// TIA Portal V20 export
// export: Created 2025-12-01T14:57:26.0447833Z, ExportSetting None, DisplayName Totally Integrated Automation Portal, DisplayVersion V20 Update 3, DisplayName TIA Portal Openness, DisplayVersion V20 Update 3, DisplayName TIA Portal Version Control Interface, DisplayVersion V20 Update 3, DisplayName STEP 7 Professional, DisplayVersion V20 Update 3, DisplayName STEP 7 Safety, DisplayVersion V20 Update 2, DisplayName WinCC Basic/Comfort/Advanced, DisplayVersion V20 Update 3, DisplayName WinCC Professional, DisplayVersion V20 Update 3, DisplayName WinCC Unified, DisplayVersion V20 Update 3
FUNCTION_BLOCK "FB454_CRTL_FRAT_E1_S2S3S4"   // FB454, LAD
TITLE = Control del Ramal de Salidas
{ S7_Optimized_Access := 'FALSE' }
AUTHOR : TLigero
NAME : 20190911
VERSION : 3.5
// stored: AutoNumber false, SetENOAutomatically false
   VAR_INPUT
      Mesa : UInt;   // Número de mesa
      En_Tension : Bool;
      pHsMx_E1 : Bool;   // pHs de ausencia de la Mesa por E1
      pHsMx_S2 : Bool;   // pHs de ausencia de la Mesa por S2
      pHsMx_S3 : Bool;   // pHs de ausencia de la Mesa por S3
      pHsMx_S4 : Bool;
      pHsMx_Pres : Bool;
      PosTR_E1S3 : Bool;   // Posicion del TR en E1E3
      PosTR_S2S4 : Bool;   // Posicion del TR en E2E4
      Termico_E1S3 : Bool;   // Proteccion del Tx en E1E3
      Termico_S2S4 : Bool;   // Proteccion del Tx en E2E4
      Avance_E1 : Bool;   // Avance del Tx en E1E3
      Avance_S2 : Bool;   // Avance del Tx en E2E4
      PTF_Sal_M2 : Bool;   // S2 >> Mesa Siguiente PTF
      NXT_Avance_S2 : Bool;   // S2 >> Mesa Siguiente avanzando
      PTF_Sal_M3 : Bool;   // S3 >> Mesa Siguiente PTF
      NXT_Avance_S3 : Bool;   // S3 >> Mesa Siguiente avanzando
      PTF_Sal_M4 : Bool;   // S2 >> Mesa Siguiente PTF
      NXT_Avance_S4 : Bool;   // S2 >> Mesa Siguiente avanzando
      F_EnvMens_Mx : Bool;   // Fin de Envio de Mensaje
      Salida_S2S4_Ausencia : Bool;   // True por ausencia. false por presencia
      Mx_BloqActivo_S2 : Bool;   // Bloqueo Activo de la Mesa
      Mx_FlujoPrin_S2 : Bool;   // El flujo principal es Saliendo por S2
      Mx_BloqActivo_S4 : Bool;   // Bloqueo Activo de la Mesa
      Mx_FlujoPrin_S4 : Bool;   // El flujo principal es Saliendo por S2
      AVTF_MAnt_Mx : Bool;   // E1 >> Mesa Anterior AVTF
      Simul_Mx : Bool;   // Activar simultaneo de mesa
      Num_Cruce : UInt;   // Número de cruce.
      DB_FIFO_Cruce : UInt := 213;   // DB de la FIFO de ordenes del cruce
      Long_FIFO_Cruce : UInt := 1;   // Longitut de la FIFO de ordenes del cruce
      ValorOrden_S2 : Word := 16#81;   // Con que orden entra por S2
      ValorOrden_S4 : Word := 16#81;   // Con que orden entra por S2
      MesaS2 : UInt;   // Número de mesa por S2
      MesaS3 : UInt;   // Número de mesa por S3
      MesaS4 : UInt;   // Número de mesa por S3
      V_CNT_ApHsMx_E1 : UDInt;   // Valor de Ausencia por E1 en ms
      V_CNT_ApHsMx_S2 : UDInt;   // Valor de Ausencia por S2 en ms
      V_CNT_ApHsMx_S3 : UDInt;   // Valor de Ausencia por S3 en ms
      V_CNT_ApHsMx_S4 : UDInt;   // Valor de Ausencia por S3 en ms
      V_CNT_SIMUL_S3 : UDInt;   // Valor de ventana para iniciar simultanero por S3 en ms
      V_Vaciado : UDInt := 15000;   // Valor de vaciado en ms
      V_TOut_Tx_Mx : UDInt := 15000;   // TimeOut de Atasco en ms
      V_TOut_TR : UDInt := 5000;   // TimeOut de Transfer en ms
   END_VAR
   VAR_OUTPUT
      P_EnvMens_PMx : Bool;   // Permiso de Enviar Mensaje de Presencia
      Etiqueta_Jdt : ULInt;   // Etiqueta que ha sido leida
      Orden_Ejecutada_Jdt : UInt;   // Orden que se ha ejecutado
      PTF_MAnt_Mx : Bool;   // E1 >> Mesa Anterior PTF
      AVTF_Sal_M2 : Bool;   // S2 >> Mesa Siguiente AVTF
      AVTF_Sal_M3 : Bool;   // S3 >> Mesa Siguiente AVTF
      AVTF_Sal_M4 : Bool;   // S3 >> Mesa Siguiente AVTF
   END_VAR
   VAR
      T1_ET00 : Bool;
      T1_ET01 : Bool;
      T1_ET02 : Bool;
      T1_ET03 : Bool;
      T1_ET10 : Bool;
      T1_ET11 : Bool;
      T1_ET12 : Bool;
      T1_ET50 : Bool;
      T1_ET60 : Bool;
      T1_ET80 : Bool;
      T1_ET70 : Bool;
      T1_ET110 : Bool;
      T1_ET111 : Bool;
      T1_ET112 : Bool;
      FIFO_OK : Bool;
      TRANS_OK : Bool;
      O_Bloqueo : Bool;
      Err_Detec_PHS : Bool;
      FN_ET02 : Bool;
      MemFN_pHsE1 : Bool;
      MemFN_pHsS3 : Bool;
      MemFN_pHsS2 : Bool;
      MemFN_pHsS4 : Bool;
      MemAuxFN_pHsE1 : Bool;
      MemAuxFN_pHsS3 : Bool;
      MemAuxFN_pHsS2 : Bool;
      MemAuxFN_pHsS4 : Bool;
      OK_TmpAusE1 : Bool;
      OK_TmpAusS3 : Bool;
      OK_TmpAusS2 : Bool;
      OK_TmpAusS4 : Bool;
      OK_Tmp_Paro : Bool;
      OK_Tmp_Simul : Bool;
      maux_fp_disparo : Bool;
      vaciado_ok { ExternalAccessible := 'False'; ExternalVisible := 'False'; ExternalWritable := 'False'} : Bool;
      Fin_reposicionamiento : Bool;
      Maux_reposicionamiento : Bool;
      CNT_Seguridad_E1 { ExternalAccessible := 'False'; ExternalVisible := 'False'; ExternalWritable := 'False'} : Bool;
      Mem_Motor_E1_Ha_Parado_NoHayPTFS2 : Bool;   // No hay permiso de transferencia a la salida por 2, por tanto cuando se reanude la secuencia a Etapa 60, no poner en marcha El motor E1
      Reposicionamiento_ok : Bool;
      TmpAus_E1 : UDInt;
      TmpAus_S2 : UDInt;
      TmpAus_S3 : UDInt;
      TmpAus_S4 : UDInt;
      TmpSeg_E1 : UDInt;
      Tmp_Paro : UDInt;
      Tmp_Simul_S3 : UDInt;
      TOUT_TR_PosS2 : UDInt;
      TOUT_TR_PosE1S3 : UDInt;
      TIM_Vaciado : UDInt;
      TOUT_E1S3 : UDInt;
      TOUT_S2 : UDInt;
      TMP_Reposicionamiento : UDInt;
      Tout_tope : UDInt;
      TMP_RearmePosicionamiento : UDInt;
      Datos_Scanner { S7_SetPoint := 'True'} : "ROUT_Orden_Fifo_Scanner";
   END_VAR
   VAR_TEMP
      O_Sal_S3 : Bool;
      O_Sal_S2 : Bool;
      O_Sal_S4 : Bool;
      O_Vaciar : Bool;
      Moti_ERRO : Bool;
      Moti_NENC : Bool;
      Moti_NORM : Bool;
      Moti_INIC : Bool;
      tout_ir_s2 : Bool;
      tout_ir_s3 : Bool;
      atasco : Bool;
      timeout_s2 : Bool;
      Tout_tope_Q : Bool;
      Aux_W_Moti : Word;
      INT_ORDEN : UInt;
      Aux_W_Orden : Word;
      I_Ord_Filtrada : UInt;
      I_V_Ord_S2 : UInt;
      I_V_Ord_S4 : UInt;
   END_VAR
   VAR_TEMP   // added for the SCL form of the ladder/FBD networks
      _w1 : Bool;
      _w2 : Bool;
      _w3 : Bool;
      _w4 : Bool;
      _w5 : Bool;
      _w6 : Bool;
   END_VAR
BEGIN

REGION Network 1: Reset Error Mesa y estado manual
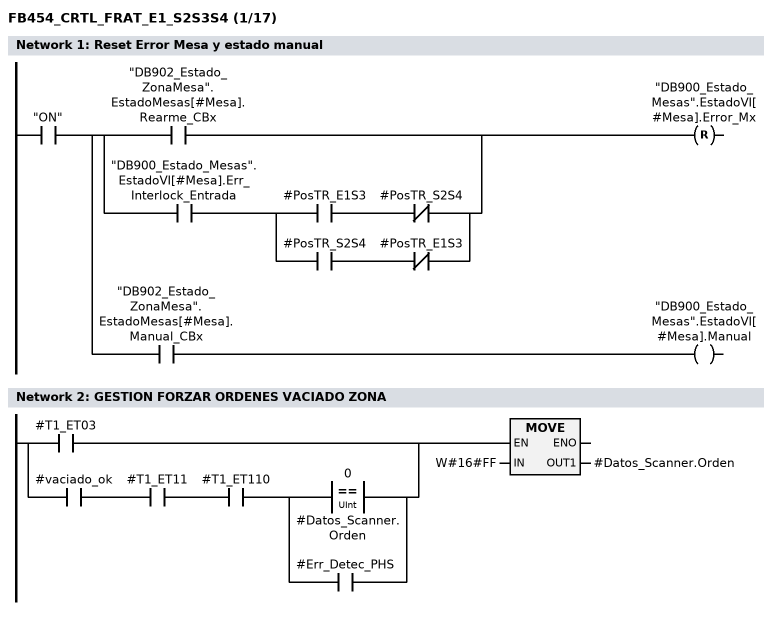
   RUNG wire#powerrail
      Contact( "ON" )
      wire#w1
      Contact( "DB902_Estado_ZonaMesa".EstadoMesas[#Mesa].Rearme_CBx )
      wire#w2
      R_Coil( "DB900_Estado_Mesas".EstadoVI[#Mesa].Error_Mx )
   END_RUNG
   RUNG wire#w1
      Contact( "DB900_Estado_Mesas".EstadoVI[#Mesa].Err_Interlock_Entrada )
      wire#w3
      Contact( #PosTR_E1S3 )
      I_Contact( #PosTR_S2S4 )
   END_RUNG wire#w2
   RUNG wire#w3
      Contact( #PosTR_S2S4 )
      I_Contact( #PosTR_E1S3 )
   END_RUNG wire#w2
   RUNG wire#w1
      Contact( "DB902_Estado_ZonaMesa".EstadoMesas[#Mesa].Manual_CBx )
      Coil( "DB900_Estado_Mesas".EstadoVI[#Mesa].Manual )
   END_RUNG
   // the same network as SCL:
   IF "ON" AND ("DB902_Estado_ZonaMesa".EstadoMesas[#Mesa].Rearme_CBx OR ("DB900_Estado_Mesas".EstadoVI[#Mesa].Err_Interlock_Entrada AND ((#PosTR_E1S3 AND NOT #PosTR_S2S4) OR (#PosTR_S2S4 AND NOT #PosTR_E1S3)))) THEN
       "DB900_Estado_Mesas".EstadoVI[#Mesa].Error_Mx := FALSE;
   END_IF;
   "DB900_Estado_Mesas".EstadoVI[#Mesa].Manual := "ON" AND "DB902_Estado_ZonaMesa".EstadoMesas[#Mesa].Manual_CBx;
END_REGION

REGION Network 2: GESTION FORZAR ORDENES VACIADO ZONA
   RUNG wire#powerrail
      Contact( #T1_ET03 )
      wire#w1
      { S7_GenerateENO := "TRUE" } Move(in := W#16#FF, out1 => #Datos_Scanner.Orden)
   END_RUNG
   RUNG wire#powerrail
      Contact( #vaciado_ok )
      Contact( #T1_ET11 )
      Contact( #T1_ET110 )
      wire#w2
      { S7_Templates := "SrcType := UInt" } EQ_Contact(in1 := 0, in2 := #Datos_Scanner.Orden)
   END_RUNG wire#w1
   RUNG wire#w2
      Contact( #Err_Detec_PHS )
   END_RUNG wire#w1
   // the same network as SCL:
   IF #T1_ET03 OR (#vaciado_ok AND #T1_ET11 AND #T1_ET110 AND ((0 = #Datos_Scanner.Orden) OR #Err_Detec_PHS)) THEN
       #Datos_Scanner.Orden := W#16#FF;
   END_IF;
END_REGION

REGION Network 3: Extraer orden
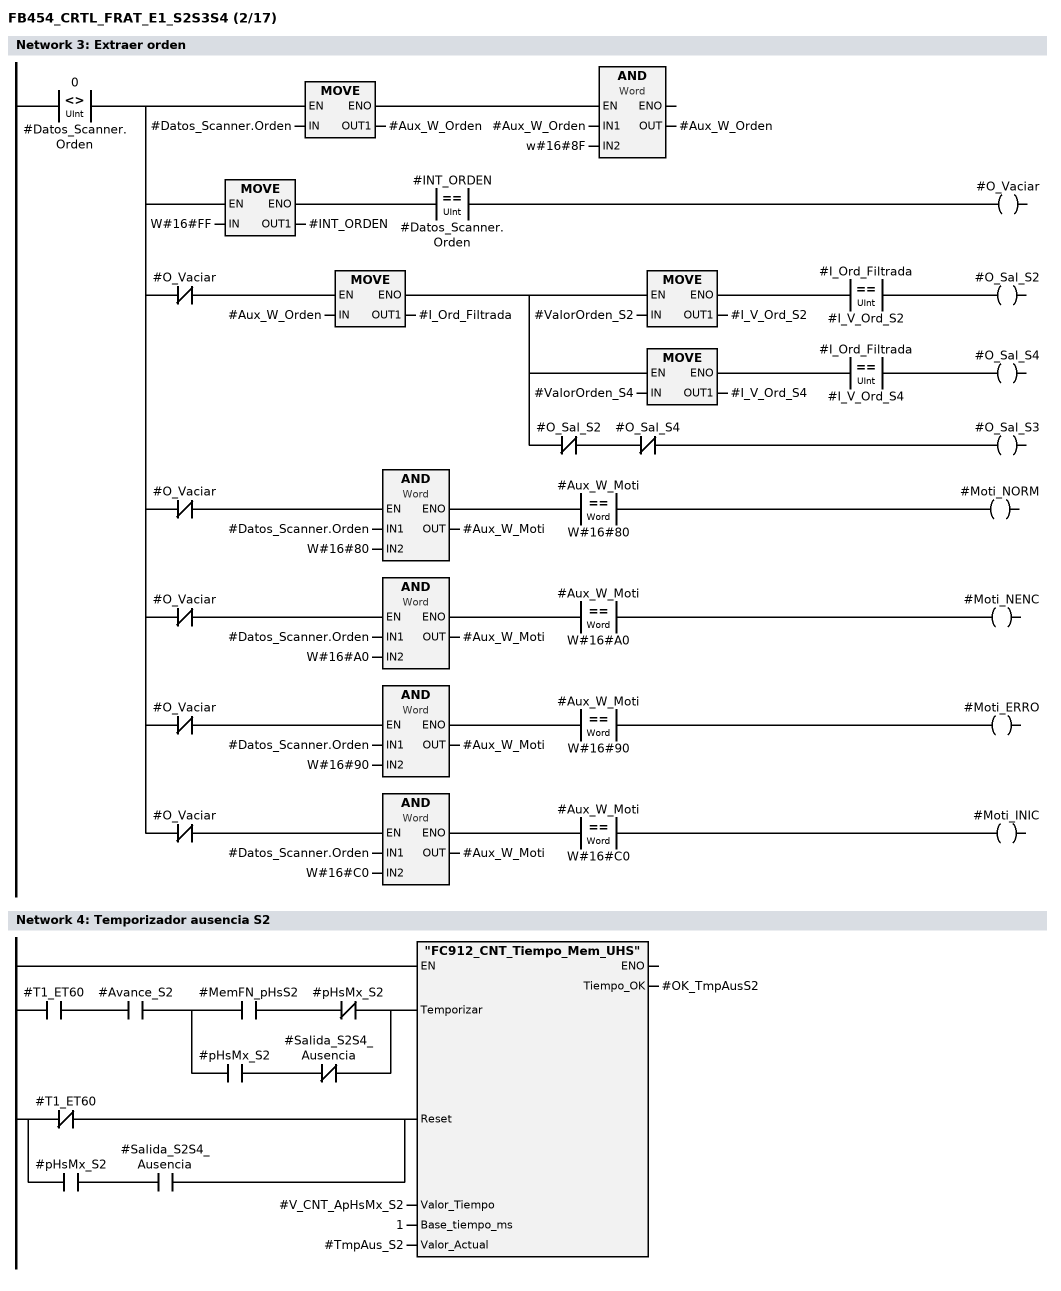
   RUNG wire#powerrail
      { S7_Templates := "SrcType := UInt" } NE_Contact(in1 := 0, in2 := #Datos_Scanner.Orden)
      wire#w1
      { S7_GenerateENO := "TRUE" } Move(in := #Datos_Scanner.Orden, out1 => #Aux_W_Orden)
      { S7_Templates := "SrcType := Word"; S7_GenerateENO := "TRUE" } And(in1 := #Aux_W_Orden, in2 := w#16#8F, out => #Aux_W_Orden)
   END_RUNG
   RUNG wire#w1
      { S7_GenerateENO := "TRUE" } Move(in := W#16#FF, out1 => #INT_ORDEN)
      { S7_Templates := "SrcType := UInt" } EQ_Contact(in1 := #INT_ORDEN, in2 := #Datos_Scanner.Orden)
      Coil( #O_Vaciar )
   END_RUNG
   RUNG wire#w1
      I_Contact( #O_Vaciar )
      { S7_GenerateENO := "TRUE" } Move(in := #Aux_W_Orden, out1 => #I_Ord_Filtrada)
      wire#w2
      { S7_GenerateENO := "TRUE" } Move(in := #ValorOrden_S2, out1 => #I_V_Ord_S2)
      { S7_Templates := "SrcType := UInt" } EQ_Contact(in1 := #I_Ord_Filtrada, in2 := #I_V_Ord_S2)
      Coil( #O_Sal_S2 )
   END_RUNG
   RUNG wire#w2
      { S7_GenerateENO := "TRUE" } Move(in := #ValorOrden_S4, out1 => #I_V_Ord_S4)
      { S7_Templates := "SrcType := UInt" } EQ_Contact(in1 := #I_Ord_Filtrada, in2 := #I_V_Ord_S4)
      Coil( #O_Sal_S4 )
   END_RUNG
   RUNG wire#w2
      I_Contact( #O_Sal_S2 )
      I_Contact( #O_Sal_S4 )
      Coil( #O_Sal_S3 )
   END_RUNG
   RUNG wire#w1
      I_Contact( #O_Vaciar )
      { S7_Templates := "SrcType := Word"; S7_GenerateENO := "TRUE" } And(in1 := #Datos_Scanner.Orden, in2 := W#16#80, out => #Aux_W_Moti)
      { S7_Templates := "SrcType := Word" } EQ_Contact(in1 := #Aux_W_Moti, in2 := W#16#80)
      Coil( #Moti_NORM )
   END_RUNG
   RUNG wire#w1
      I_Contact( #O_Vaciar )
      { S7_Templates := "SrcType := Word"; S7_GenerateENO := "TRUE" } And(in1 := #Datos_Scanner.Orden, in2 := W#16#A0, out => #Aux_W_Moti)
      { S7_Templates := "SrcType := Word" } EQ_Contact(in1 := #Aux_W_Moti, in2 := W#16#A0)
      Coil( #Moti_NENC )
   END_RUNG
   RUNG wire#w1
      I_Contact( #O_Vaciar )
      { S7_Templates := "SrcType := Word"; S7_GenerateENO := "TRUE" } And(in1 := #Datos_Scanner.Orden, in2 := W#16#90, out => #Aux_W_Moti)
      { S7_Templates := "SrcType := Word" } EQ_Contact(in1 := #Aux_W_Moti, in2 := W#16#90)
      Coil( #Moti_ERRO )
   END_RUNG
   RUNG wire#w1
      I_Contact( #O_Vaciar )
      { S7_Templates := "SrcType := Word"; S7_GenerateENO := "TRUE" } And(in1 := #Datos_Scanner.Orden, in2 := W#16#C0, out => #Aux_W_Moti)
      { S7_Templates := "SrcType := Word" } EQ_Contact(in1 := #Aux_W_Moti, in2 := W#16#C0)
      Coil( #Moti_INIC )
   END_RUNG
   // the same network as SCL:
   // ENO of a box is taken as its EN; it also drops when the box reports an error
   #_w1 := 0 <> #Datos_Scanner.Orden;
   IF #_w1 THEN
       #Aux_W_Orden := #Datos_Scanner.Orden;
       #Aux_W_Orden := #Aux_W_Orden AND w#16#8F;
       #INT_ORDEN := W#16#FF;
   END_IF;
   #O_Vaciar := #_w1 AND (#INT_ORDEN = #Datos_Scanner.Orden);
   #_w2 := #_w1 AND NOT #O_Vaciar;
   IF #_w2 THEN
       #I_Ord_Filtrada := #Aux_W_Orden;
       #I_V_Ord_S2 := #ValorOrden_S2;
   END_IF;
   #O_Sal_S2 := #_w2 AND (#I_Ord_Filtrada = #I_V_Ord_S2);
   IF #_w2 THEN #I_V_Ord_S4 := #ValorOrden_S4; END_IF;
   #O_Sal_S4 := #_w2 AND (#I_Ord_Filtrada = #I_V_Ord_S4);
   #O_Sal_S3 := #_w2 AND NOT #O_Sal_S2 AND NOT #O_Sal_S4;
   #_w3 := #_w1 AND NOT #O_Vaciar;
   IF #_w3 THEN #Aux_W_Moti := #Datos_Scanner.Orden AND W#16#80; END_IF;
   #Moti_NORM := #_w3 AND (#Aux_W_Moti = W#16#80);
   #_w4 := #_w1 AND NOT #O_Vaciar;
   IF #_w4 THEN #Aux_W_Moti := #Datos_Scanner.Orden AND W#16#A0; END_IF;
   #Moti_NENC := #_w4 AND (#Aux_W_Moti = W#16#A0);
   #_w5 := #_w1 AND NOT #O_Vaciar;
   IF #_w5 THEN #Aux_W_Moti := #Datos_Scanner.Orden AND W#16#90; END_IF;
   #Moti_ERRO := #_w5 AND (#Aux_W_Moti = W#16#90);
   #_w6 := #_w1 AND NOT #O_Vaciar;
   IF #_w6 THEN #Aux_W_Moti := #Datos_Scanner.Orden AND W#16#C0; END_IF;
   #Moti_INIC := #_w6 AND (#Aux_W_Moti = W#16#C0);
END_REGION

REGION Network 4: Temporizador ausencia S2
   RUNG wire#powerrail
      "FC912_CNT_Tiempo_Mem_UHS"(Temporizar := wire#w2, Reset := wire#w3, Valor_Tiempo := #V_CNT_ApHsMx_S2, Base_tiempo_ms := 1, Valor_Actual := #TmpAus_S2, Tiempo_OK => #OK_TmpAusS2)
   END_RUNG
   RUNG wire#powerrail
      Contact( #T1_ET60 )
      Contact( #Avance_S2 )
      wire#w1
      Contact( #MemFN_pHsS2 )
      I_Contact( #pHsMx_S2 )
   END_RUNG wire#w2
   RUNG wire#w1
      Contact( #pHsMx_S2 )
      I_Contact( #Salida_S2S4_Ausencia )
   END_RUNG wire#w2
   RUNG wire#powerrail
      I_Contact( #T1_ET60 )
   END_RUNG wire#w3
   RUNG wire#powerrail
      Contact( #pHsMx_S2 )
      Contact( #Salida_S2S4_Ausencia )
   END_RUNG wire#w3
   // the same network as SCL:
   "FC912_CNT_Tiempo_Mem_UHS"(Temporizar := #T1_ET60 AND #Avance_S2 AND ((#MemFN_pHsS2 AND NOT #pHsMx_S2) OR (#pHsMx_S2 AND NOT #Salida_S2S4_Ausencia)),
                           Reset := NOT #T1_ET60 OR (#pHsMx_S2 AND #Salida_S2S4_Ausencia),
                           Valor_Tiempo := #V_CNT_ApHsMx_S2,
                           Base_tiempo_ms := 1,
                           Valor_Actual := #TmpAus_S2,
                           Tiempo_OK => #OK_TmpAusS2);
END_REGION

REGION Network 5: Temporizador ausencia S4
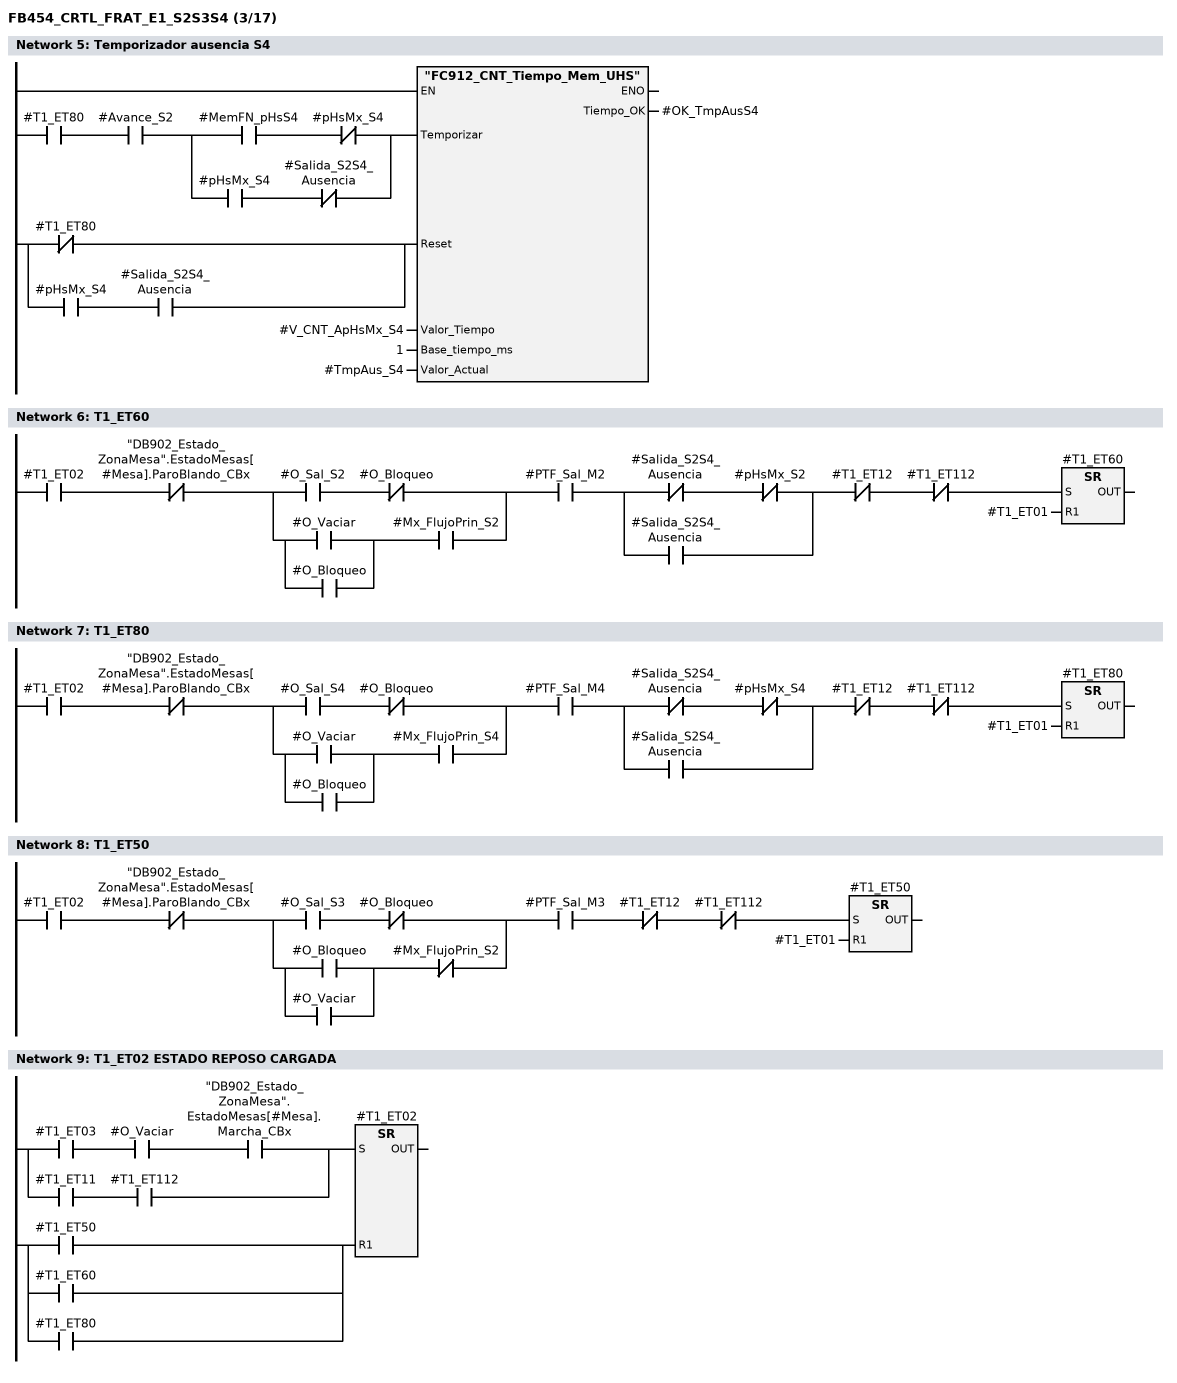
   RUNG wire#powerrail
      "FC912_CNT_Tiempo_Mem_UHS"(Temporizar := wire#w2, Reset := wire#w3, Valor_Tiempo := #V_CNT_ApHsMx_S4, Base_tiempo_ms := 1, Valor_Actual := #TmpAus_S4, Tiempo_OK => #OK_TmpAusS4)
   END_RUNG
   RUNG wire#powerrail
      Contact( #T1_ET80 )
      Contact( #Avance_S2 )
      wire#w1
      Contact( #MemFN_pHsS4 )
      I_Contact( #pHsMx_S4 )
   END_RUNG wire#w2
   RUNG wire#w1
      Contact( #pHsMx_S4 )
      I_Contact( #Salida_S2S4_Ausencia )
   END_RUNG wire#w2
   RUNG wire#powerrail
      I_Contact( #T1_ET80 )
   END_RUNG wire#w3
   RUNG wire#powerrail
      Contact( #pHsMx_S4 )
      Contact( #Salida_S2S4_Ausencia )
   END_RUNG wire#w3
   // the same network as SCL:
   "FC912_CNT_Tiempo_Mem_UHS"(Temporizar := #T1_ET80 AND #Avance_S2 AND ((#MemFN_pHsS4 AND NOT #pHsMx_S4) OR (#pHsMx_S4 AND NOT #Salida_S2S4_Ausencia)),
                           Reset := NOT #T1_ET80 OR (#pHsMx_S4 AND #Salida_S2S4_Ausencia),
                           Valor_Tiempo := #V_CNT_ApHsMx_S4,
                           Base_tiempo_ms := 1,
                           Valor_Actual := #TmpAus_S4,
                           Tiempo_OK => #OK_TmpAusS4);
END_REGION

REGION Network 6: T1_ET60
   RUNG wire#powerrail
      Contact( #T1_ET02 )
      I_Contact( "DB902_Estado_ZonaMesa".EstadoMesas[#Mesa].ParoBlando_CBx )
      wire#w1
      Contact( #O_Sal_S2 )
      I_Contact( #O_Bloqueo )
      wire#w2
      Contact( #PTF_Sal_M2 )
      wire#w4
      I_Contact( #Salida_S2S4_Ausencia )
      I_Contact( #pHsMx_S2 )
      wire#w5
      I_Contact( #T1_ET12 )
      I_Contact( #T1_ET112 )
      S_SR(operand := #T1_ET60, r1 := #T1_ET01)
   END_RUNG
   RUNG wire#w1
      Contact( #O_Vaciar )
      wire#w3
      Contact( #Mx_FlujoPrin_S2 )
   END_RUNG wire#w2
   RUNG wire#w1
      Contact( #O_Bloqueo )
   END_RUNG wire#w3
   RUNG wire#w4
      Contact( #Salida_S2S4_Ausencia )
   END_RUNG wire#w5
   // the same network as SCL:
   IF #T1_ET02 AND NOT "DB902_Estado_ZonaMesa".EstadoMesas[#Mesa].ParoBlando_CBx AND ((#O_Sal_S2 AND NOT #O_Bloqueo) OR ((#O_Vaciar OR #O_Bloqueo) AND #Mx_FlujoPrin_S2)) AND #PTF_Sal_M2 AND ((NOT #Salida_S2S4_Ausencia AND NOT #pHsMx_S2) OR #Salida_S2S4_Ausencia) AND NOT #T1_ET12 AND NOT #T1_ET112 THEN
       #T1_ET60 := TRUE;   // SR flip-flop
   END_IF;
   IF #T1_ET01 THEN #T1_ET60 := FALSE; END_IF;
END_REGION

REGION Network 7: T1_ET80
   RUNG wire#powerrail
      Contact( #T1_ET02 )
      I_Contact( "DB902_Estado_ZonaMesa".EstadoMesas[#Mesa].ParoBlando_CBx )
      wire#w1
      Contact( #O_Sal_S4 )
      I_Contact( #O_Bloqueo )
      wire#w2
      Contact( #PTF_Sal_M4 )
      wire#w4
      I_Contact( #Salida_S2S4_Ausencia )
      I_Contact( #pHsMx_S4 )
      wire#w5
      I_Contact( #T1_ET12 )
      I_Contact( #T1_ET112 )
      S_SR(operand := #T1_ET80, r1 := #T1_ET01)
   END_RUNG
   RUNG wire#w1
      Contact( #O_Vaciar )
      wire#w3
      Contact( #Mx_FlujoPrin_S4 )
   END_RUNG wire#w2
   RUNG wire#w1
      Contact( #O_Bloqueo )
   END_RUNG wire#w3
   RUNG wire#w4
      Contact( #Salida_S2S4_Ausencia )
   END_RUNG wire#w5
   // the same network as SCL:
   IF #T1_ET02 AND NOT "DB902_Estado_ZonaMesa".EstadoMesas[#Mesa].ParoBlando_CBx AND ((#O_Sal_S4 AND NOT #O_Bloqueo) OR ((#O_Vaciar OR #O_Bloqueo) AND #Mx_FlujoPrin_S4)) AND #PTF_Sal_M4 AND ((NOT #Salida_S2S4_Ausencia AND NOT #pHsMx_S4) OR #Salida_S2S4_Ausencia) AND NOT #T1_ET12 AND NOT #T1_ET112 THEN
       #T1_ET80 := TRUE;   // SR flip-flop
   END_IF;
   IF #T1_ET01 THEN #T1_ET80 := FALSE; END_IF;
END_REGION

REGION Network 8: T1_ET50
   RUNG wire#powerrail
      Contact( #T1_ET02 )
      I_Contact( "DB902_Estado_ZonaMesa".EstadoMesas[#Mesa].ParoBlando_CBx )
      wire#w1
      Contact( #O_Sal_S3 )
      I_Contact( #O_Bloqueo )
      wire#w2
      Contact( #PTF_Sal_M3 )
      I_Contact( #T1_ET12 )
      I_Contact( #T1_ET112 )
      S_SR(operand := #T1_ET50, r1 := #T1_ET01)
   END_RUNG
   RUNG wire#w1
      Contact( #O_Bloqueo )
      wire#w3
      I_Contact( #Mx_FlujoPrin_S2 )
   END_RUNG wire#w2
   RUNG wire#w1
      Contact( #O_Vaciar )
   END_RUNG wire#w3
   // the same network as SCL:
   IF #T1_ET02 AND NOT "DB902_Estado_ZonaMesa".EstadoMesas[#Mesa].ParoBlando_CBx AND ((#O_Sal_S3 AND NOT #O_Bloqueo) OR ((#O_Bloqueo OR #O_Vaciar) AND NOT #Mx_FlujoPrin_S2)) AND #PTF_Sal_M3 AND NOT #T1_ET12 AND NOT #T1_ET112 THEN
       #T1_ET50 := TRUE;   // SR flip-flop
   END_IF;
   IF #T1_ET01 THEN #T1_ET50 := FALSE; END_IF;
END_REGION

REGION Network 9: T1_ET02 ESTADO REPOSO CARGADA
   RUNG wire#powerrail
      Contact( #T1_ET03 )
      Contact( #O_Vaciar )
      Contact( "DB902_Estado_ZonaMesa".EstadoMesas[#Mesa].Marcha_CBx )
      wire#w1
      S_SR(operand := #T1_ET02, r1 := wire#w2)
   END_RUNG
   RUNG wire#powerrail
      Contact( #T1_ET11 )
      Contact( #T1_ET112 )
   END_RUNG wire#w1
   RUNG wire#powerrail
      Contact( #T1_ET50 )
   END_RUNG wire#w2
   RUNG wire#powerrail
      Contact( #T1_ET60 )
   END_RUNG wire#w2
   RUNG wire#powerrail
      Contact( #T1_ET80 )
   END_RUNG wire#w2
   // the same network as SCL:
   IF (#T1_ET03 AND #O_Vaciar AND "DB902_Estado_ZonaMesa".EstadoMesas[#Mesa].Marcha_CBx) OR (#T1_ET11 AND #T1_ET112) THEN
       #T1_ET02 := TRUE;   // SR flip-flop
   END_IF;
   IF #T1_ET50 OR #T1_ET60 OR #T1_ET80 THEN #T1_ET02 := FALSE; END_IF;
END_REGION

REGION Network 10: T1_ET03 RESET
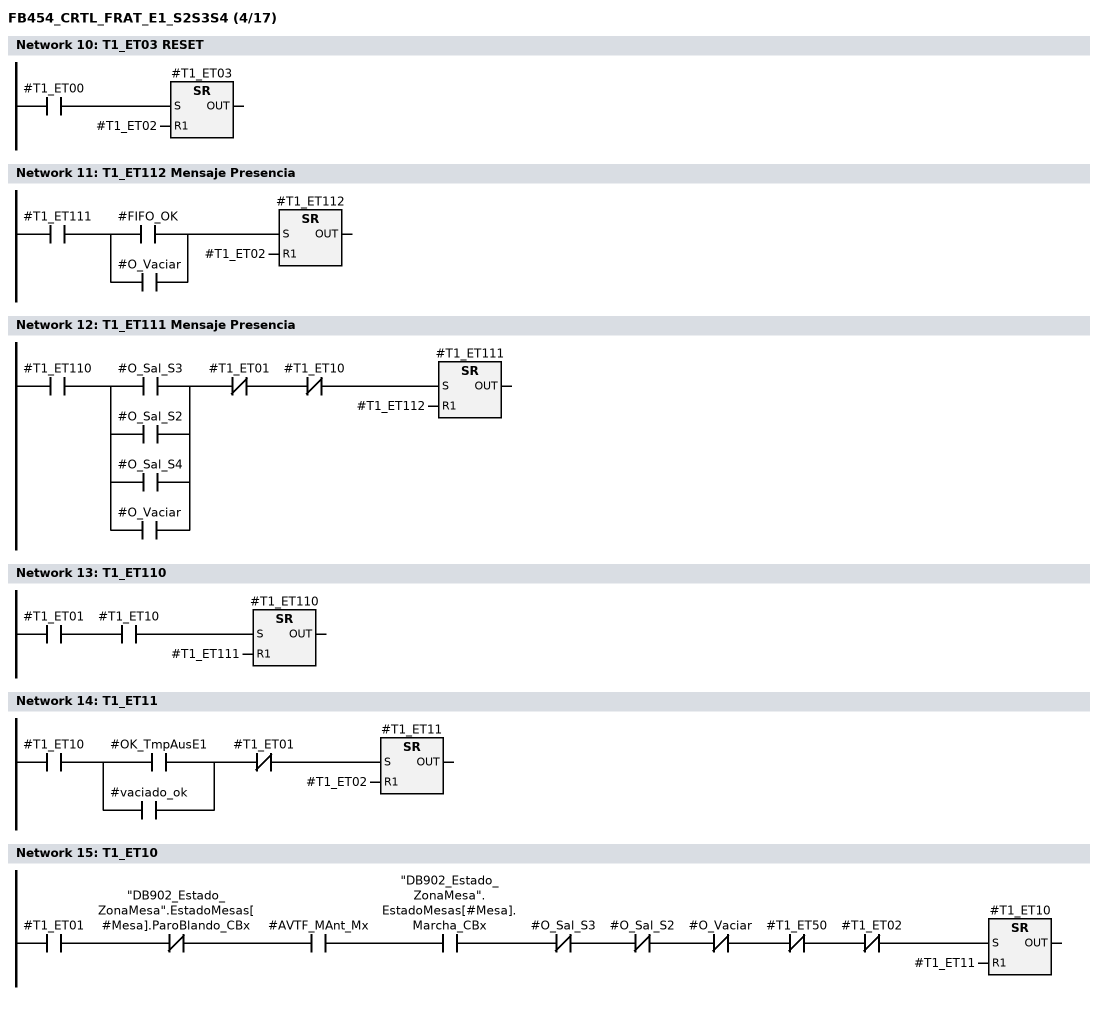
   RUNG wire#powerrail
      Contact( #T1_ET00 )
      S_SR(operand := #T1_ET03, r1 := #T1_ET02)
   END_RUNG
   // the same network as SCL:
   IF #T1_ET00 THEN
       #T1_ET03 := TRUE;   // SR flip-flop
   END_IF;
   IF #T1_ET02 THEN #T1_ET03 := FALSE; END_IF;
END_REGION

REGION Network 11: T1_ET112 Mensaje Presencia
   RUNG wire#powerrail
      Contact( #T1_ET111 )
      wire#w1
      Contact( #FIFO_OK )
      wire#w2
      S_SR(operand := #T1_ET112, r1 := #T1_ET02)
   END_RUNG
   RUNG wire#w1
      Contact( #O_Vaciar )
   END_RUNG wire#w2
   // the same network as SCL:
   IF #T1_ET111 AND (#FIFO_OK OR #O_Vaciar) THEN
       #T1_ET112 := TRUE;   // SR flip-flop
   END_IF;
   IF #T1_ET02 THEN #T1_ET112 := FALSE; END_IF;
END_REGION

REGION Network 12: T1_ET111 Mensaje Presencia
   RUNG wire#powerrail
      Contact( #T1_ET110 )
      wire#w1
      Contact( #O_Sal_S3 )
      wire#w2
      I_Contact( #T1_ET01 )
      I_Contact( #T1_ET10 )
      S_SR(operand := #T1_ET111, r1 := #T1_ET112)
   END_RUNG
   RUNG wire#w1
      Contact( #O_Sal_S2 )
   END_RUNG wire#w2
   RUNG wire#w1
      Contact( #O_Sal_S4 )
   END_RUNG wire#w2
   RUNG wire#w1
      Contact( #O_Vaciar )
   END_RUNG wire#w2
   // the same network as SCL:
   IF #T1_ET110 AND (#O_Sal_S3 OR #O_Sal_S2 OR #O_Sal_S4 OR #O_Vaciar) AND NOT #T1_ET01 AND NOT #T1_ET10 THEN
       #T1_ET111 := TRUE;   // SR flip-flop
   END_IF;
   IF #T1_ET112 THEN #T1_ET111 := FALSE; END_IF;
END_REGION

REGION Network 13: T1_ET110
   RUNG wire#powerrail
      Contact( #T1_ET01 )
      Contact( #T1_ET10 )
      S_SR(operand := #T1_ET110, r1 := #T1_ET111)
   END_RUNG
   // the same network as SCL:
   IF #T1_ET01 AND #T1_ET10 THEN
       #T1_ET110 := TRUE;   // SR flip-flop
   END_IF;
   IF #T1_ET111 THEN #T1_ET110 := FALSE; END_IF;
END_REGION

REGION Network 14: T1_ET11
   RUNG wire#powerrail
      Contact( #T1_ET10 )
      wire#w1
      Contact( #OK_TmpAusE1 )
      wire#w2
      I_Contact( #T1_ET01 )
      S_SR(operand := #T1_ET11, r1 := #T1_ET02)
   END_RUNG
   RUNG wire#w1
      Contact( #vaciado_ok )
   END_RUNG wire#w2
   // the same network as SCL:
   IF #T1_ET10 AND (#OK_TmpAusE1 OR #vaciado_ok) AND NOT #T1_ET01 THEN
       #T1_ET11 := TRUE;   // SR flip-flop
   END_IF;
   IF #T1_ET02 THEN #T1_ET11 := FALSE; END_IF;
END_REGION

REGION Network 15: T1_ET10
   RUNG wire#powerrail
      Contact( #T1_ET01 )
      I_Contact( "DB902_Estado_ZonaMesa".EstadoMesas[#Mesa].ParoBlando_CBx )
      Contact( #AVTF_MAnt_Mx )
      Contact( "DB902_Estado_ZonaMesa".EstadoMesas[#Mesa].Marcha_CBx )
      I_Contact( #O_Sal_S3 )
      I_Contact( #O_Sal_S2 )
      I_Contact( #O_Vaciar )
      I_Contact( #T1_ET50 )
      I_Contact( #T1_ET02 )
      S_SR(operand := #T1_ET10, r1 := #T1_ET11)
   END_RUNG
   // the same network as SCL:
   IF #T1_ET01 AND NOT "DB902_Estado_ZonaMesa".EstadoMesas[#Mesa].ParoBlando_CBx AND #AVTF_MAnt_Mx AND "DB902_Estado_ZonaMesa".EstadoMesas[#Mesa].Marcha_CBx AND NOT #O_Sal_S3 AND NOT #O_Sal_S2 AND NOT #O_Vaciar AND NOT #T1_ET50 AND NOT #T1_ET02 THEN
       #T1_ET10 := TRUE;   // SR flip-flop
   END_IF;
   IF #T1_ET11 THEN #T1_ET10 := FALSE; END_IF;
END_REGION

REGION Network 16: T1_ET01 ESTADO REPOSO VACIO
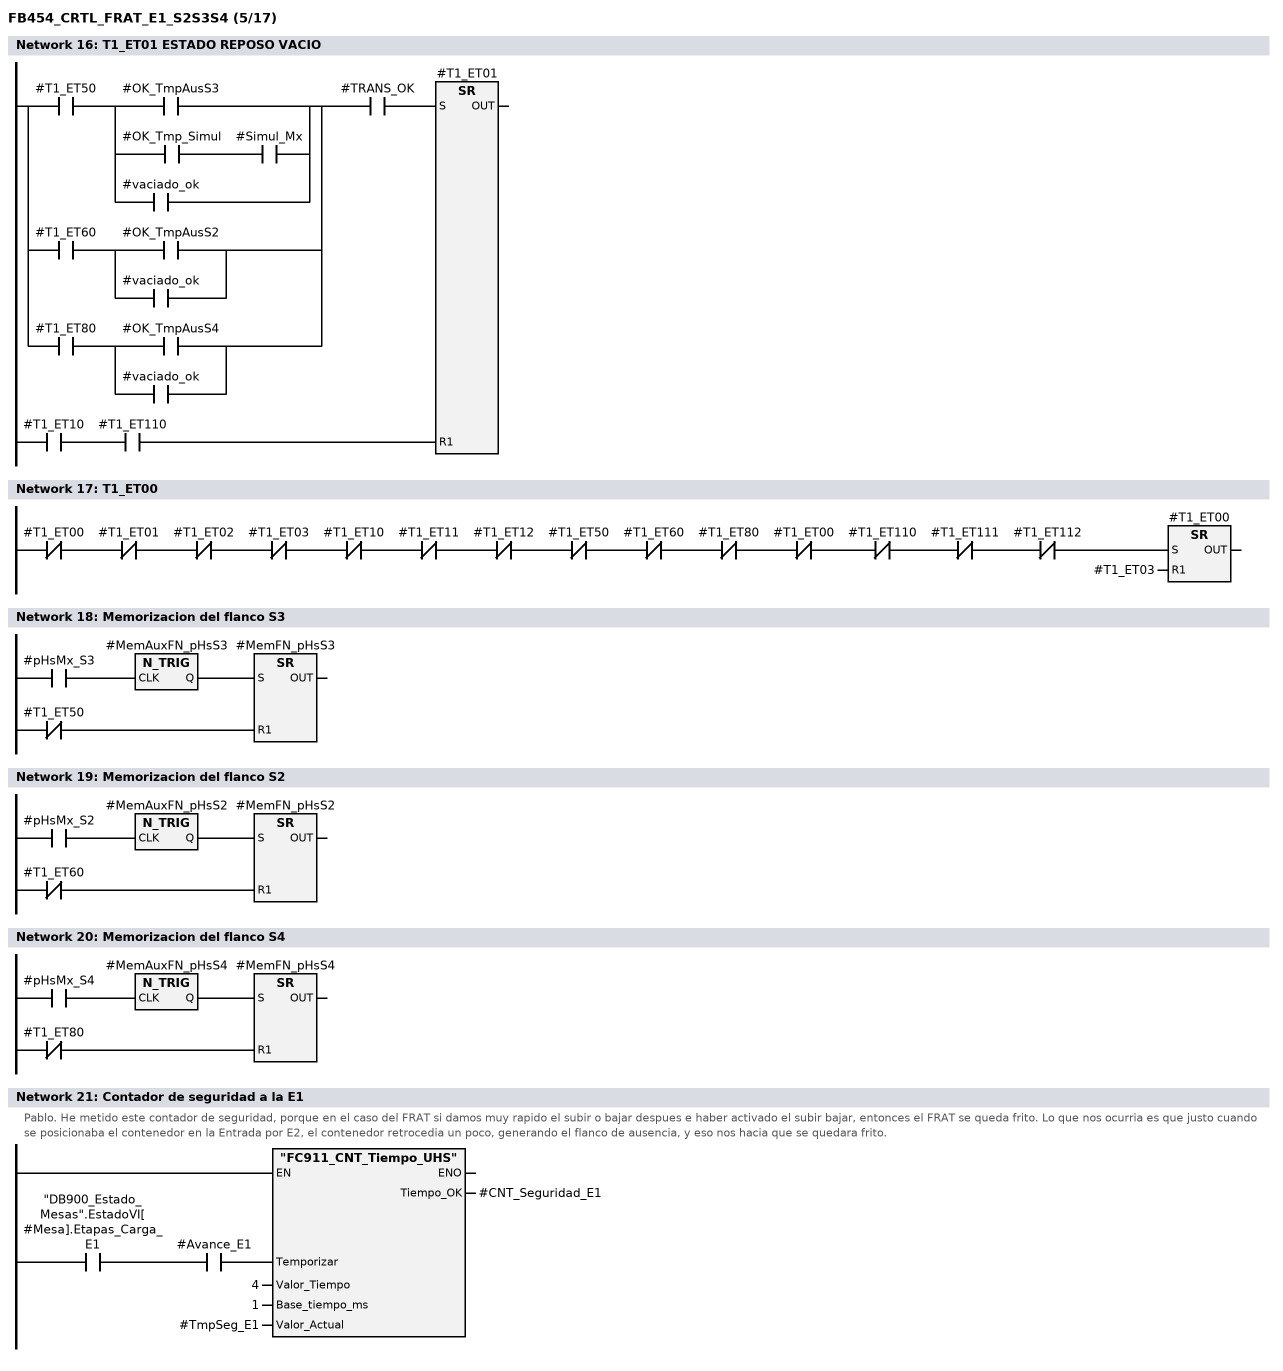
   RUNG wire#powerrail
      Contact( #T1_ET50 )
      wire#w1
      Contact( #OK_TmpAusS3 )
      wire#w2
      Contact( #TRANS_OK )
      S_SR(operand := #T1_ET01, r1 := wire#w5)
   END_RUNG
   RUNG wire#w1
      Contact( #OK_Tmp_Simul )
      Contact( #Simul_Mx )
   END_RUNG wire#w2
   RUNG wire#w1
      Contact( #vaciado_ok )
   END_RUNG wire#w2
   RUNG wire#powerrail
      Contact( #T1_ET60 )
      wire#w3
      Contact( #OK_TmpAusS2 )
   END_RUNG wire#w2
   RUNG wire#w3
      Contact( #vaciado_ok )
   END_RUNG wire#w2
   RUNG wire#powerrail
      Contact( #T1_ET80 )
      wire#w4
      Contact( #OK_TmpAusS4 )
   END_RUNG wire#w2
   RUNG wire#w4
      Contact( #vaciado_ok )
   END_RUNG wire#w2
   RUNG wire#powerrail
      Contact( #T1_ET10 )
      Contact( #T1_ET110 )
   END_RUNG wire#w5
   // the same network as SCL:
   IF ((#T1_ET50 AND (#OK_TmpAusS3 OR (#OK_Tmp_Simul AND #Simul_Mx) OR #vaciado_ok)) OR (#T1_ET60 AND (#OK_TmpAusS2 OR #vaciado_ok)) OR (#T1_ET80 AND (#OK_TmpAusS4 OR #vaciado_ok))) AND #TRANS_OK THEN
       #T1_ET01 := TRUE;   // SR flip-flop
   END_IF;
   IF #T1_ET10 AND #T1_ET110 THEN #T1_ET01 := FALSE; END_IF;
END_REGION

REGION Network 17: T1_ET00
   RUNG wire#powerrail
      I_Contact( #T1_ET00 )
      I_Contact( #T1_ET01 )
      I_Contact( #T1_ET02 )
      I_Contact( #T1_ET03 )
      I_Contact( #T1_ET10 )
      I_Contact( #T1_ET11 )
      I_Contact( #T1_ET12 )
      I_Contact( #T1_ET50 )
      I_Contact( #T1_ET60 )
      I_Contact( #T1_ET80 )
      I_Contact( #T1_ET00 )
      I_Contact( #T1_ET110 )
      I_Contact( #T1_ET111 )
      I_Contact( #T1_ET112 )
      S_SR(operand := #T1_ET00, r1 := #T1_ET03)
   END_RUNG
   // the same network as SCL:
   IF NOT #T1_ET00 AND NOT #T1_ET01 AND NOT #T1_ET02 AND NOT #T1_ET03 AND NOT #T1_ET10 AND NOT #T1_ET11 AND NOT #T1_ET12 AND NOT #T1_ET50 AND NOT #T1_ET60 AND NOT #T1_ET80 AND NOT #T1_ET00 AND NOT #T1_ET110 AND NOT #T1_ET111 AND NOT #T1_ET112 THEN
       #T1_ET00 := TRUE;   // SR flip-flop
   END_IF;
   IF #T1_ET03 THEN #T1_ET00 := FALSE; END_IF;
END_REGION

REGION Network 18: Memorizacion del flanco S3
   RUNG wire#powerrail
      Contact( #pHsMx_S3 )
      N_Trig( #MemAuxFN_pHsS3 )
      S_SR(operand := #MemFN_pHsS3, r1 := wire#w1)
   END_RUNG
   RUNG wire#powerrail
      I_Contact( #T1_ET50 )
   END_RUNG wire#w1
   // the same network as SCL:
   #_w1 := NOT #pHsMx_S3 AND #MemAuxFN_pHsS3;   // falling edge
   #MemAuxFN_pHsS3 := #pHsMx_S3;
   IF #_w1 THEN
       #MemFN_pHsS3 := TRUE;   // SR flip-flop
   END_IF;
   IF NOT #T1_ET50 THEN #MemFN_pHsS3 := FALSE; END_IF;
END_REGION

REGION Network 19: Memorizacion del flanco S2
   RUNG wire#powerrail
      Contact( #pHsMx_S2 )
      N_Trig( #MemAuxFN_pHsS2 )
      S_SR(operand := #MemFN_pHsS2, r1 := wire#w1)
   END_RUNG
   RUNG wire#powerrail
      I_Contact( #T1_ET60 )
   END_RUNG wire#w1
   // the same network as SCL:
   #_w1 := NOT #pHsMx_S2 AND #MemAuxFN_pHsS2;   // falling edge
   #MemAuxFN_pHsS2 := #pHsMx_S2;
   IF #_w1 THEN
       #MemFN_pHsS2 := TRUE;   // SR flip-flop
   END_IF;
   IF NOT #T1_ET60 THEN #MemFN_pHsS2 := FALSE; END_IF;
END_REGION

REGION Network 20: Memorizacion del flanco S4
   RUNG wire#powerrail
      Contact( #pHsMx_S4 )
      N_Trig( #MemAuxFN_pHsS4 )
      S_SR(operand := #MemFN_pHsS4, r1 := wire#w1)
   END_RUNG
   RUNG wire#powerrail
      I_Contact( #T1_ET80 )
   END_RUNG wire#w1
   // the same network as SCL:
   #_w1 := NOT #pHsMx_S4 AND #MemAuxFN_pHsS4;   // falling edge
   #MemAuxFN_pHsS4 := #pHsMx_S4;
   IF #_w1 THEN
       #MemFN_pHsS4 := TRUE;   // SR flip-flop
   END_IF;
   IF NOT #T1_ET80 THEN #MemFN_pHsS4 := FALSE; END_IF;
END_REGION

REGION Network 21: Contador de seguridad a la E1
   // Pablo. He metido este contador de seguridad, porque en el caso del FRAT si damos muy rapido el subir o bajar despues e haber activado el subir bajar, entonces el FRAT se queda frito. Lo que nos ocurria es que justo cuando se posicionaba el contenedor en la Entrada por E2, el contenedor retrocedia un poco, generando el flanco de ausencia, y eso nos hacia que se quedara frito.
   RUNG wire#powerrail
      "FC911_CNT_Tiempo_UHS"(Temporizar := wire#w1, Valor_Tiempo := 4, Base_tiempo_ms := 1, Valor_Actual := #TmpSeg_E1, Tiempo_OK => #CNT_Seguridad_E1)
   END_RUNG
   RUNG wire#powerrail
      Contact( "DB900_Estado_Mesas".EstadoVI[#Mesa].Etapas_Carga_E1 )
      Contact( #Avance_E1 )
   END_RUNG wire#w1
   // the same network as SCL:
   "FC911_CNT_Tiempo_UHS"(Temporizar := "DB900_Estado_Mesas".EstadoVI[#Mesa].Etapas_Carga_E1 AND #Avance_E1,
                          Valor_Tiempo := 4,
                          Base_tiempo_ms := 1,
                          Valor_Actual := #TmpSeg_E1,
                          Tiempo_OK => #CNT_Seguridad_E1);
END_REGION

REGION Network 22: Memorizacion del flanco E1
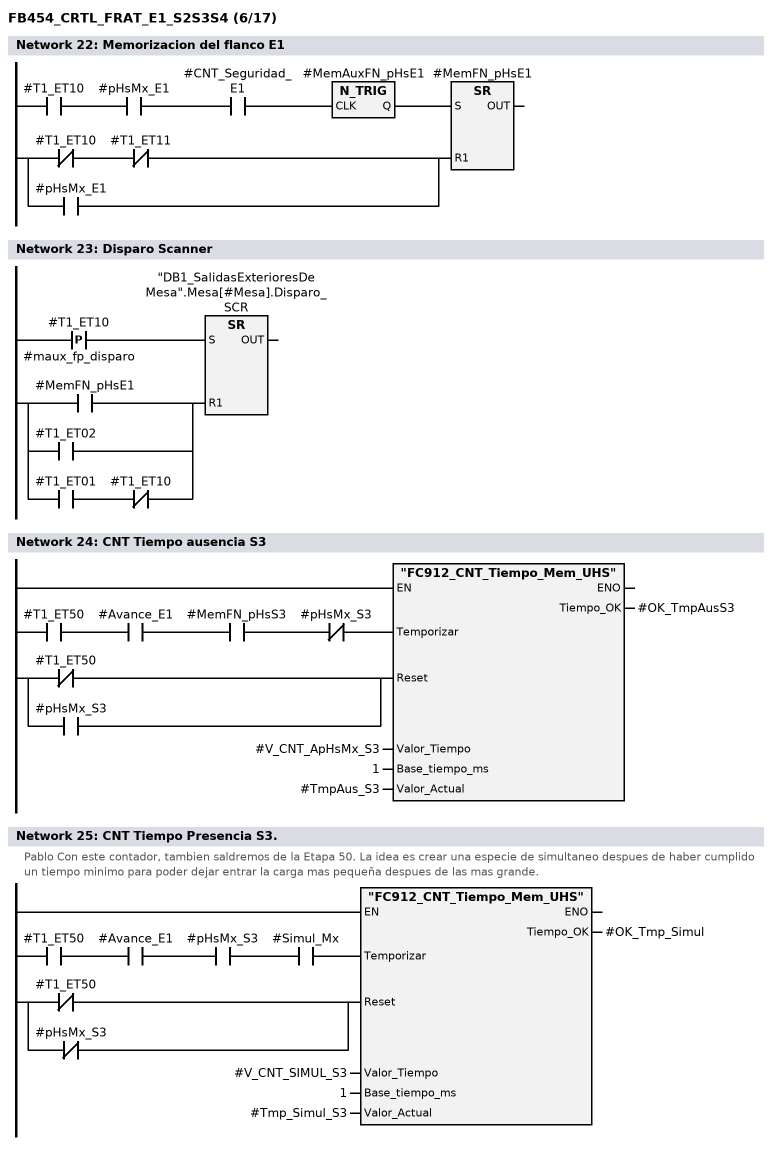
   RUNG wire#powerrail
      Contact( #T1_ET10 )
      Contact( #pHsMx_E1 )
      Contact( #CNT_Seguridad_E1 )
      N_Trig( #MemAuxFN_pHsE1 )
      S_SR(operand := #MemFN_pHsE1, r1 := wire#w1)
   END_RUNG
   RUNG wire#powerrail
      I_Contact( #T1_ET10 )
      I_Contact( #T1_ET11 )
   END_RUNG wire#w1
   RUNG wire#powerrail
      Contact( #pHsMx_E1 )
   END_RUNG wire#w1
   // the same network as SCL:
   #_w1 := #T1_ET10 AND #pHsMx_E1 AND #CNT_Seguridad_E1;
   #_w2 := NOT #_w1 AND #MemAuxFN_pHsE1;   // falling edge
   #MemAuxFN_pHsE1 := #_w1;
   IF #_w2 THEN
       #MemFN_pHsE1 := TRUE;   // SR flip-flop
   END_IF;
   IF (NOT #T1_ET10 AND NOT #T1_ET11) OR #pHsMx_E1 THEN #MemFN_pHsE1 := FALSE; END_IF;
END_REGION

REGION Network 23: Disparo Scanner
   RUNG wire#powerrail
      P_Contact(operand := #T1_ET10, bit := #maux_fp_disparo)
      S_SR(operand := "DB1_SalidasExterioresDeMesa".Mesa[#Mesa].Disparo_SCR, r1 := wire#w1)
   END_RUNG
   RUNG wire#powerrail
      Contact( #MemFN_pHsE1 )
   END_RUNG wire#w1
   RUNG wire#powerrail
      Contact( #T1_ET02 )
   END_RUNG wire#w1
   RUNG wire#powerrail
      Contact( #T1_ET01 )
      I_Contact( #T1_ET10 )
   END_RUNG wire#w1
   // the same network as SCL:
   #_w1 := #T1_ET10 AND NOT #maux_fp_disparo;   // rising edge of #T1_ET10
   #maux_fp_disparo := #T1_ET10;
   IF #_w1 THEN
       "DB1_SalidasExterioresDeMesa".Mesa[#Mesa].Disparo_SCR := TRUE;   // SR flip-flop
   END_IF;
   IF #MemFN_pHsE1 OR #T1_ET02 OR (#T1_ET01 AND NOT #T1_ET10) THEN
       "DB1_SalidasExterioresDeMesa".Mesa[#Mesa].Disparo_SCR := FALSE;
   END_IF;
END_REGION

REGION Network 24: CNT Tiempo ausencia S3
   RUNG wire#powerrail
      "FC912_CNT_Tiempo_Mem_UHS"(Temporizar := wire#w1, Reset := wire#w2, Valor_Tiempo := #V_CNT_ApHsMx_S3, Base_tiempo_ms := 1, Valor_Actual := #TmpAus_S3, Tiempo_OK => #OK_TmpAusS3)
   END_RUNG
   RUNG wire#powerrail
      Contact( #T1_ET50 )
      Contact( #Avance_E1 )
      Contact( #MemFN_pHsS3 )
      I_Contact( #pHsMx_S3 )
   END_RUNG wire#w1
   RUNG wire#powerrail
      I_Contact( #T1_ET50 )
   END_RUNG wire#w2
   RUNG wire#powerrail
      Contact( #pHsMx_S3 )
   END_RUNG wire#w2
   // the same network as SCL:
   "FC912_CNT_Tiempo_Mem_UHS"(Temporizar := #T1_ET50 AND #Avance_E1 AND #MemFN_pHsS3 AND NOT #pHsMx_S3,
                           Reset := NOT #T1_ET50 OR #pHsMx_S3,
                           Valor_Tiempo := #V_CNT_ApHsMx_S3,
                           Base_tiempo_ms := 1,
                           Valor_Actual := #TmpAus_S3,
                           Tiempo_OK => #OK_TmpAusS3);
END_REGION

REGION Network 25: CNT Tiempo Presencia S3.
   // Pablo Con este contador, tambien saldremos de la Etapa 50. La idea es crear una especie de simultaneo despues de haber cumplido un tiempo minimo para poder dejar entrar la carga mas pequeña despues de las mas grande.
   RUNG wire#powerrail
      "FC912_CNT_Tiempo_Mem_UHS"(Temporizar := wire#w1, Reset := wire#w2, Valor_Tiempo := #V_CNT_SIMUL_S3, Base_tiempo_ms := 1, Valor_Actual := #Tmp_Simul_S3, Tiempo_OK => #OK_Tmp_Simul)
   END_RUNG
   RUNG wire#powerrail
      Contact( #T1_ET50 )
      Contact( #Avance_E1 )
      Contact( #pHsMx_S3 )
      Contact( #Simul_Mx )
   END_RUNG wire#w1
   RUNG wire#powerrail
      I_Contact( #T1_ET50 )
   END_RUNG wire#w2
   RUNG wire#powerrail
      I_Contact( #pHsMx_S3 )
   END_RUNG wire#w2
   // the same network as SCL:
   "FC912_CNT_Tiempo_Mem_UHS"(Temporizar := #T1_ET50 AND #Avance_E1 AND #pHsMx_S3 AND #Simul_Mx,
                           Reset := NOT #T1_ET50 OR NOT #pHsMx_S3,
                           Valor_Tiempo := #V_CNT_SIMUL_S3,
                           Base_tiempo_ms := 1,
                           Valor_Actual := #Tmp_Simul_S3,
                           Tiempo_OK => #OK_Tmp_Simul);
END_REGION

REGION Network 26: CNT Tiempo ausencia E1
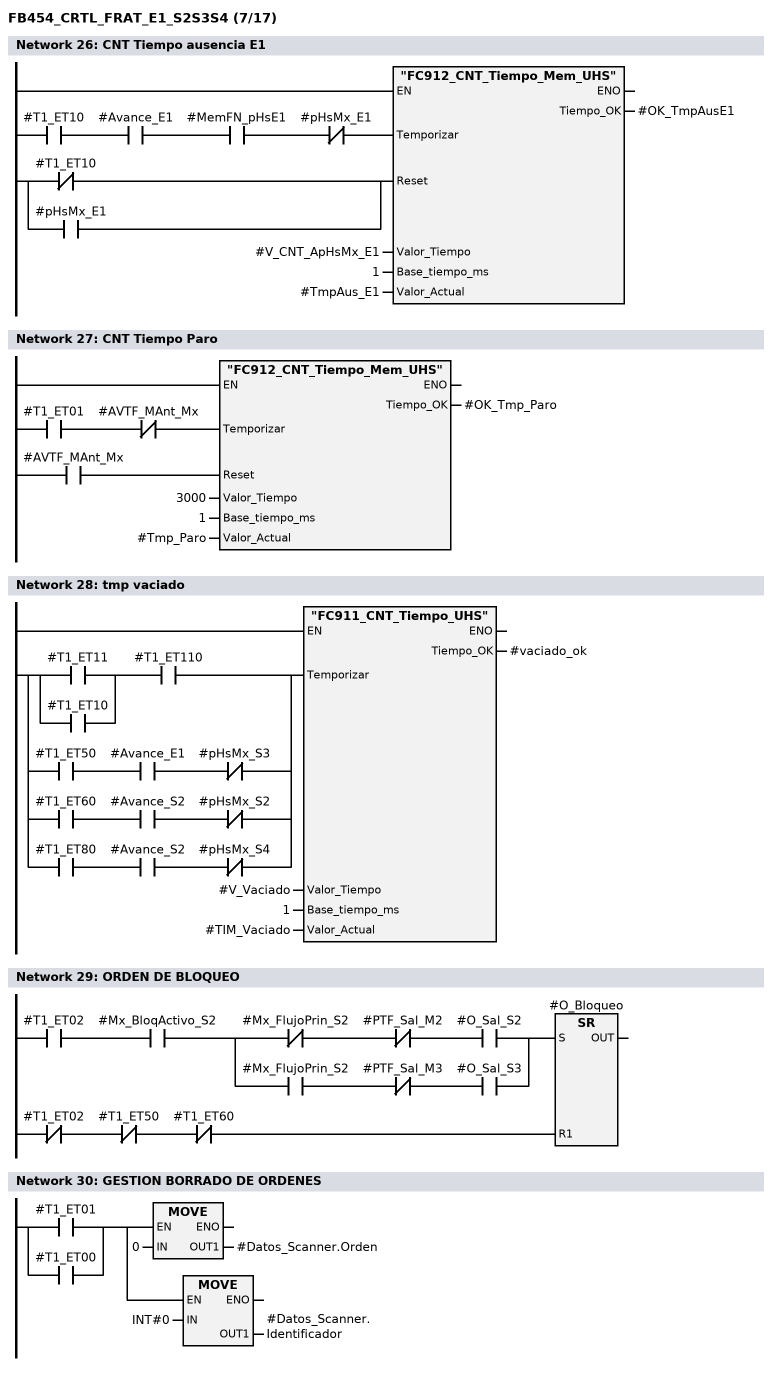
   RUNG wire#powerrail
      "FC912_CNT_Tiempo_Mem_UHS"(Temporizar := wire#w1, Reset := wire#w2, Valor_Tiempo := #V_CNT_ApHsMx_E1, Base_tiempo_ms := 1, Valor_Actual := #TmpAus_E1, Tiempo_OK => #OK_TmpAusE1)
   END_RUNG
   RUNG wire#powerrail
      Contact( #T1_ET10 )
      Contact( #Avance_E1 )
      Contact( #MemFN_pHsE1 )
      I_Contact( #pHsMx_E1 )
   END_RUNG wire#w1
   RUNG wire#powerrail
      I_Contact( #T1_ET10 )
   END_RUNG wire#w2
   RUNG wire#powerrail
      Contact( #pHsMx_E1 )
   END_RUNG wire#w2
   // the same network as SCL:
   "FC912_CNT_Tiempo_Mem_UHS"(Temporizar := #T1_ET10 AND #Avance_E1 AND #MemFN_pHsE1 AND NOT #pHsMx_E1,
                           Reset := NOT #T1_ET10 OR #pHsMx_E1,
                           Valor_Tiempo := #V_CNT_ApHsMx_E1,
                           Base_tiempo_ms := 1,
                           Valor_Actual := #TmpAus_E1,
                           Tiempo_OK => #OK_TmpAusE1);
END_REGION

REGION Network 27: CNT Tiempo Paro
   RUNG wire#powerrail
      "FC912_CNT_Tiempo_Mem_UHS"(Temporizar := wire#w1, Reset := wire#w2, Valor_Tiempo := 3000, Base_tiempo_ms := 1, Valor_Actual := #Tmp_Paro, Tiempo_OK => #OK_Tmp_Paro)
   END_RUNG
   RUNG wire#powerrail
      Contact( #T1_ET01 )
      I_Contact( #AVTF_MAnt_Mx )
   END_RUNG wire#w1
   RUNG wire#powerrail
      Contact( #AVTF_MAnt_Mx )
   END_RUNG wire#w2
   // the same network as SCL:
   "FC912_CNT_Tiempo_Mem_UHS"(Temporizar := #T1_ET01 AND NOT #AVTF_MAnt_Mx,
                           Reset := #AVTF_MAnt_Mx,
                           Valor_Tiempo := 3000,
                           Base_tiempo_ms := 1,
                           Valor_Actual := #Tmp_Paro,
                           Tiempo_OK => #OK_Tmp_Paro);
END_REGION

REGION Network 28: tmp vaciado
   RUNG wire#powerrail
      "FC911_CNT_Tiempo_UHS"(Temporizar := wire#w2, Valor_Tiempo := #V_Vaciado, Base_tiempo_ms := 1, Valor_Actual := #TIM_Vaciado, Tiempo_OK => #vaciado_ok)
   END_RUNG
   RUNG wire#powerrail
      Contact( #T1_ET11 )
      wire#w1
      Contact( #T1_ET110 )
   END_RUNG wire#w2
   RUNG wire#powerrail
      Contact( #T1_ET10 )
   END_RUNG wire#w1
   RUNG wire#powerrail
      Contact( #T1_ET50 )
      Contact( #Avance_E1 )
      I_Contact( #pHsMx_S3 )
   END_RUNG wire#w2
   RUNG wire#powerrail
      Contact( #T1_ET60 )
      Contact( #Avance_S2 )
      I_Contact( #pHsMx_S2 )
   END_RUNG wire#w2
   RUNG wire#powerrail
      Contact( #T1_ET80 )
      Contact( #Avance_S2 )
      I_Contact( #pHsMx_S4 )
   END_RUNG wire#w2
   // the same network as SCL:
   "FC911_CNT_Tiempo_UHS"(Temporizar := ((#T1_ET11 OR #T1_ET10) AND #T1_ET110) OR (#T1_ET50 AND #Avance_E1 AND NOT #pHsMx_S3) OR (#T1_ET60 AND #Avance_S2 AND NOT #pHsMx_S2) OR (#T1_ET80 AND #Avance_S2 AND NOT #pHsMx_S4),
                          Valor_Tiempo := #V_Vaciado,
                          Base_tiempo_ms := 1,
                          Valor_Actual := #TIM_Vaciado,
                          Tiempo_OK => #vaciado_ok);
END_REGION

REGION Network 29: ORDEN DE BLOQUEO
   RUNG wire#powerrail
      Contact( #T1_ET02 )
      Contact( #Mx_BloqActivo_S2 )
      wire#w1
      I_Contact( #Mx_FlujoPrin_S2 )
      I_Contact( #PTF_Sal_M2 )
      Contact( #O_Sal_S2 )
      wire#w2
      S_SR(operand := #O_Bloqueo, r1 := wire#w3)
   END_RUNG
   RUNG wire#w1
      Contact( #Mx_FlujoPrin_S2 )
      I_Contact( #PTF_Sal_M3 )
      Contact( #O_Sal_S3 )
   END_RUNG wire#w2
   RUNG wire#powerrail
      I_Contact( #T1_ET02 )
      I_Contact( #T1_ET50 )
      I_Contact( #T1_ET60 )
   END_RUNG wire#w3
   // the same network as SCL:
   IF #T1_ET02 AND #Mx_BloqActivo_S2 AND ((NOT #Mx_FlujoPrin_S2 AND NOT #PTF_Sal_M2 AND #O_Sal_S2) OR (#Mx_FlujoPrin_S2 AND NOT #PTF_Sal_M3 AND #O_Sal_S3)) THEN
       #O_Bloqueo := TRUE;   // SR flip-flop
   END_IF;
   IF NOT #T1_ET02 AND NOT #T1_ET50 AND NOT #T1_ET60 THEN #O_Bloqueo := FALSE; END_IF;
END_REGION

REGION Network 30: GESTION BORRADO DE ORDENES
   RUNG wire#powerrail
      Contact( #T1_ET01 )
      wire#w1
      { S7_GenerateENO := "TRUE" } Move(in := 0, out1 => #Datos_Scanner.Orden)
   END_RUNG
   RUNG wire#powerrail
      Contact( #T1_ET00 )
   END_RUNG wire#w1
   RUNG wire#w1
      { S7_GenerateENO := "TRUE" } Move(in := INT#0, out1 => #Datos_Scanner.Identificador)
   END_RUNG
   // the same network as SCL:
   IF #T1_ET01 OR #T1_ET00 THEN
       #Datos_Scanner.Orden := 0;
       #Datos_Scanner.Identificador := INT#0;
   END_IF;
END_REGION

REGION Network 31: TOMA ORDENES FIFO
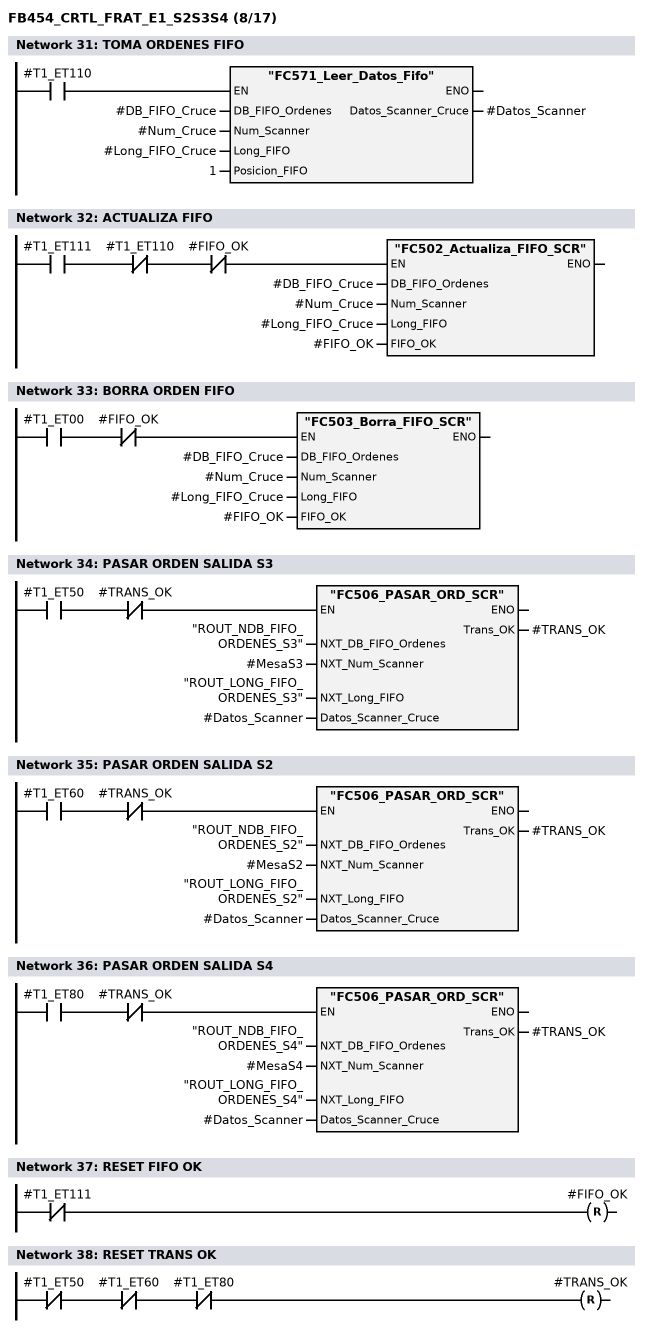
   RUNG wire#powerrail
      Contact( #T1_ET110 )
      "FC571_Leer_Datos_Fifo"(DB_FIFO_Ordenes := #DB_FIFO_Cruce, Num_Scanner := #Num_Cruce, Long_FIFO := #Long_FIFO_Cruce, Posicion_FIFO := 1, Datos_Scanner_Cruce => #Datos_Scanner)
   END_RUNG
   // the same network as SCL:
   IF #T1_ET110 THEN
       "FC571_Leer_Datos_Fifo"(DB_FIFO_Ordenes := #DB_FIFO_Cruce,
                               Num_Scanner := #Num_Cruce,
                               Long_FIFO := #Long_FIFO_Cruce,
                               Posicion_FIFO := 1,
                               Datos_Scanner_Cruce => #Datos_Scanner);
   END_IF;
END_REGION

REGION Network 32: ACTUALIZA FIFO
   RUNG wire#powerrail
      Contact( #T1_ET111 )
      I_Contact( #T1_ET110 )
      I_Contact( #FIFO_OK )
      "FC502_Actualiza_FIFO_SCR"(DB_FIFO_Ordenes := #DB_FIFO_Cruce, Num_Scanner := #Num_Cruce, Long_FIFO := #Long_FIFO_Cruce, FIFO_OK := #FIFO_OK)
   END_RUNG
   // the same network as SCL:
   IF #T1_ET111 AND NOT #T1_ET110 AND NOT #FIFO_OK THEN
       "FC502_Actualiza_FIFO_SCR"(DB_FIFO_Ordenes := #DB_FIFO_Cruce,
                               Num_Scanner := #Num_Cruce,
                               Long_FIFO := #Long_FIFO_Cruce,
                               FIFO_OK := #FIFO_OK);
   END_IF;
END_REGION

REGION Network 33: BORRA ORDEN FIFO
   RUNG wire#powerrail
      Contact( #T1_ET00 )
      I_Contact( #FIFO_OK )
      "FC503_Borra_FIFO_SCR"(DB_FIFO_Ordenes := #DB_FIFO_Cruce, Num_Scanner := #Num_Cruce, Long_FIFO := #Long_FIFO_Cruce, FIFO_OK := #FIFO_OK)
   END_RUNG
   // the same network as SCL:
   IF #T1_ET00 AND NOT #FIFO_OK THEN
       "FC503_Borra_FIFO_SCR"(DB_FIFO_Ordenes := #DB_FIFO_Cruce,
                              Num_Scanner := #Num_Cruce,
                              Long_FIFO := #Long_FIFO_Cruce,
                              FIFO_OK := #FIFO_OK);
   END_IF;
END_REGION

REGION Network 34: PASAR ORDEN SALIDA S3
   RUNG wire#powerrail
      Contact( #T1_ET50 )
      I_Contact( #TRANS_OK )
      "FC506_PASAR_ORD_SCR"(NXT_DB_FIFO_Ordenes := "ROUT_NDB_FIFO_ORDENES_S3", NXT_Num_Scanner := #MesaS3, NXT_Long_FIFO := "ROUT_LONG_FIFO_ORDENES_S3", Datos_Scanner_Cruce := #Datos_Scanner, Trans_OK => #TRANS_OK)
   END_RUNG
   // the same network as SCL:
   IF #T1_ET50 AND NOT #TRANS_OK THEN
       "FC506_PASAR_ORD_SCR"(NXT_DB_FIFO_Ordenes := "ROUT_NDB_FIFO_ORDENES_S3",
                             NXT_Num_Scanner := #MesaS3,
                             NXT_Long_FIFO := "ROUT_LONG_FIFO_ORDENES_S3",
                             Datos_Scanner_Cruce := #Datos_Scanner,
                             Trans_OK => #TRANS_OK);
   END_IF;
END_REGION

REGION Network 35: PASAR ORDEN SALIDA S2
   RUNG wire#powerrail
      Contact( #T1_ET60 )
      I_Contact( #TRANS_OK )
      "FC506_PASAR_ORD_SCR"(NXT_DB_FIFO_Ordenes := "ROUT_NDB_FIFO_ORDENES_S2", NXT_Num_Scanner := #MesaS2, NXT_Long_FIFO := "ROUT_LONG_FIFO_ORDENES_S2", Datos_Scanner_Cruce := #Datos_Scanner, Trans_OK => #TRANS_OK)
   END_RUNG
   // the same network as SCL:
   IF #T1_ET60 AND NOT #TRANS_OK THEN
       "FC506_PASAR_ORD_SCR"(NXT_DB_FIFO_Ordenes := "ROUT_NDB_FIFO_ORDENES_S2",
                             NXT_Num_Scanner := #MesaS2,
                             NXT_Long_FIFO := "ROUT_LONG_FIFO_ORDENES_S2",
                             Datos_Scanner_Cruce := #Datos_Scanner,
                             Trans_OK => #TRANS_OK);
   END_IF;
END_REGION

REGION Network 36: PASAR ORDEN SALIDA S4
   RUNG wire#powerrail
      Contact( #T1_ET80 )
      I_Contact( #TRANS_OK )
      "FC506_PASAR_ORD_SCR"(NXT_DB_FIFO_Ordenes := "ROUT_NDB_FIFO_ORDENES_S4", NXT_Num_Scanner := #MesaS4, NXT_Long_FIFO := "ROUT_LONG_FIFO_ORDENES_S4", Datos_Scanner_Cruce := #Datos_Scanner, Trans_OK => #TRANS_OK)
   END_RUNG
   // the same network as SCL:
   IF #T1_ET80 AND NOT #TRANS_OK THEN
       "FC506_PASAR_ORD_SCR"(NXT_DB_FIFO_Ordenes := "ROUT_NDB_FIFO_ORDENES_S4",
                             NXT_Num_Scanner := #MesaS4,
                             NXT_Long_FIFO := "ROUT_LONG_FIFO_ORDENES_S4",
                             Datos_Scanner_Cruce := #Datos_Scanner,
                             Trans_OK => #TRANS_OK);
   END_IF;
END_REGION

REGION Network 37: RESET FIFO OK
   RUNG wire#powerrail
      I_Contact( #T1_ET111 )
      R_Coil( #FIFO_OK )
   END_RUNG
   // the same network as SCL:
   IF NOT #T1_ET111 THEN #FIFO_OK := FALSE; END_IF;
END_REGION

REGION Network 38: RESET TRANS OK
   RUNG wire#powerrail
      I_Contact( #T1_ET50 )
      I_Contact( #T1_ET60 )
      I_Contact( #T1_ET80 )
      R_Coil( #TRANS_OK )
   END_RUNG
   // the same network as SCL:
   IF NOT #T1_ET50 AND NOT #T1_ET60 AND NOT #T1_ET80 THEN #TRANS_OK := FALSE; END_IF;
END_REGION

REGION Network 39: PREVIO CARGA OK
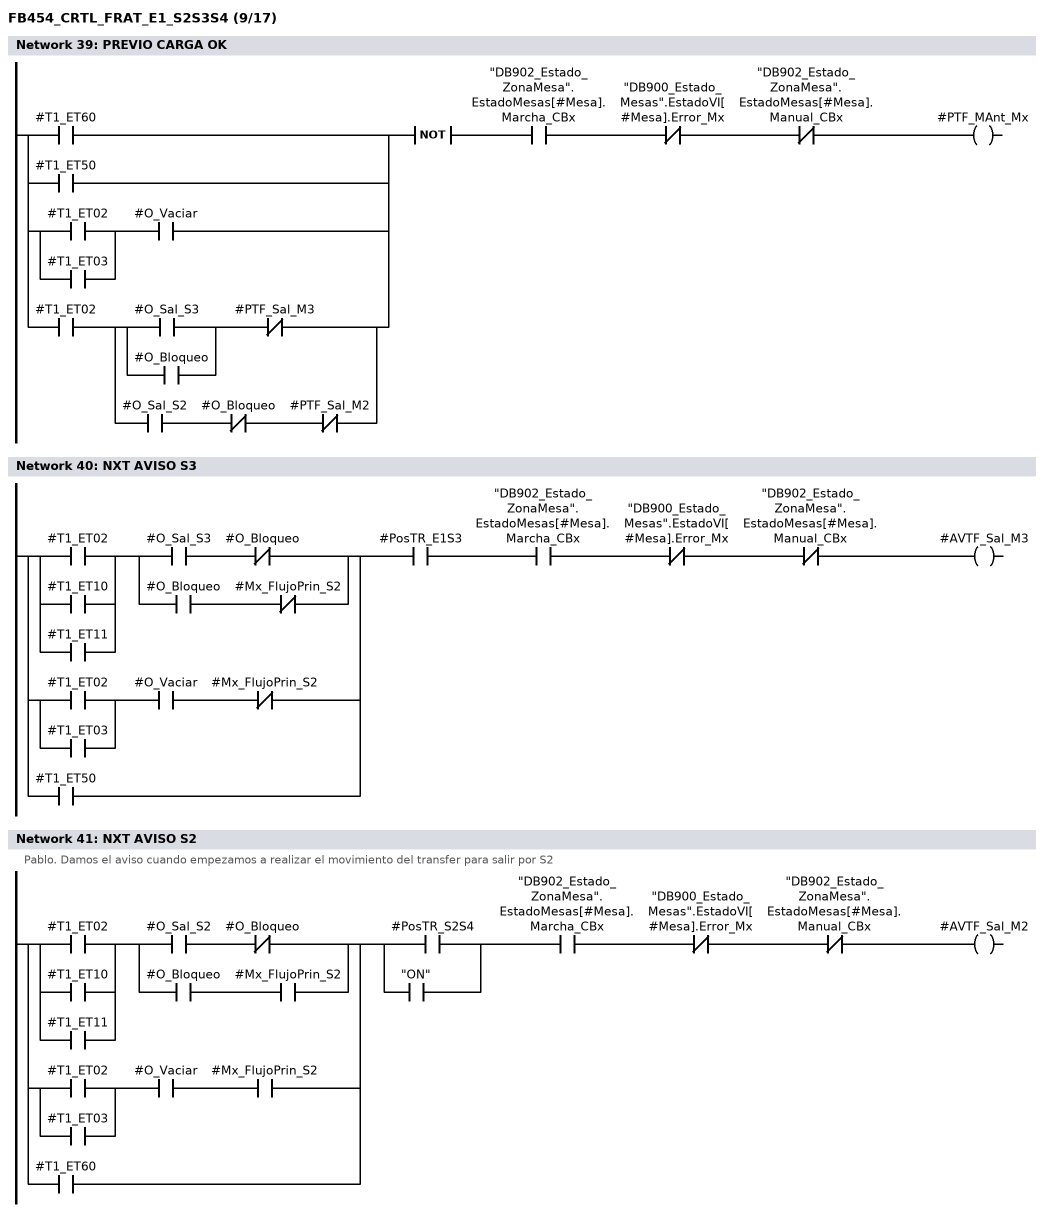
   RUNG wire#powerrail
      Contact( #T1_ET60 )
      wire#w1
      Not()
      Contact( "DB902_Estado_ZonaMesa".EstadoMesas[#Mesa].Marcha_CBx )
      I_Contact( "DB900_Estado_Mesas".EstadoVI[#Mesa].Error_Mx )
      I_Contact( "DB902_Estado_ZonaMesa".EstadoMesas[#Mesa].Manual_CBx )
      Coil( #PTF_MAnt_Mx )
   END_RUNG
   RUNG wire#powerrail
      Contact( #T1_ET50 )
   END_RUNG wire#w1
   RUNG wire#powerrail
      Contact( #T1_ET02 )
      wire#w2
      Contact( #O_Vaciar )
   END_RUNG wire#w1
   RUNG wire#powerrail
      Contact( #T1_ET03 )
   END_RUNG wire#w2
   RUNG wire#powerrail
      Contact( #T1_ET02 )
      wire#w3
      Contact( #O_Sal_S3 )
      wire#w4
      I_Contact( #PTF_Sal_M3 )
   END_RUNG wire#w1
   RUNG wire#w3
      Contact( #O_Bloqueo )
   END_RUNG wire#w4
   RUNG wire#w3
      Contact( #O_Sal_S2 )
      I_Contact( #O_Bloqueo )
      I_Contact( #PTF_Sal_M2 )
   END_RUNG wire#w1
   // the same network as SCL:
   #PTF_MAnt_Mx := NOT (#T1_ET60 OR #T1_ET50 OR ((#T1_ET02 OR #T1_ET03) AND #O_Vaciar) OR (#T1_ET02 AND (((#O_Sal_S3 OR #O_Bloqueo) AND NOT #PTF_Sal_M3) OR (#O_Sal_S2 AND NOT #O_Bloqueo AND NOT #PTF_Sal_M2)))) AND "DB902_Estado_ZonaMesa".EstadoMesas[#Mesa].Marcha_CBx AND NOT "DB900_Estado_Mesas".EstadoVI[#Mesa].Error_Mx AND NOT "DB902_Estado_ZonaMesa".EstadoMesas[#Mesa].Manual_CBx;
END_REGION

REGION Network 40: NXT AVISO S3
   RUNG wire#powerrail
      Contact( #T1_ET02 )
      wire#w1
      Contact( #O_Sal_S3 )
      I_Contact( #O_Bloqueo )
      wire#w2
      Contact( #PosTR_E1S3 )
      Contact( "DB902_Estado_ZonaMesa".EstadoMesas[#Mesa].Marcha_CBx )
      I_Contact( "DB900_Estado_Mesas".EstadoVI[#Mesa].Error_Mx )
      I_Contact( "DB902_Estado_ZonaMesa".EstadoMesas[#Mesa].Manual_CBx )
      Coil( #AVTF_Sal_M3 )
   END_RUNG
   RUNG wire#powerrail
      Contact( #T1_ET10 )
   END_RUNG wire#w1
   RUNG wire#powerrail
      Contact( #T1_ET11 )
   END_RUNG wire#w1
   RUNG wire#w1
      Contact( #O_Bloqueo )
      I_Contact( #Mx_FlujoPrin_S2 )
   END_RUNG wire#w2
   RUNG wire#powerrail
      Contact( #T1_ET02 )
      wire#w3
      Contact( #O_Vaciar )
      I_Contact( #Mx_FlujoPrin_S2 )
   END_RUNG wire#w2
   RUNG wire#powerrail
      Contact( #T1_ET03 )
   END_RUNG wire#w3
   RUNG wire#powerrail
      Contact( #T1_ET50 )
   END_RUNG wire#w2
   // the same network as SCL:
   #AVTF_Sal_M3 := (((#T1_ET02 OR #T1_ET10 OR #T1_ET11) AND ((#O_Sal_S3 AND NOT #O_Bloqueo) OR (#O_Bloqueo AND NOT #Mx_FlujoPrin_S2))) OR ((#T1_ET02 OR #T1_ET03) AND #O_Vaciar AND NOT #Mx_FlujoPrin_S2) OR #T1_ET50) AND #PosTR_E1S3 AND "DB902_Estado_ZonaMesa".EstadoMesas[#Mesa].Marcha_CBx AND NOT "DB900_Estado_Mesas".EstadoVI[#Mesa].Error_Mx AND NOT "DB902_Estado_ZonaMesa".EstadoMesas[#Mesa].Manual_CBx;
END_REGION

REGION Network 41: NXT AVISO S2
   // Pablo. Damos el aviso cuando empezamos a realizar el movimiento del transfer para salir por S2
   RUNG wire#powerrail
      Contact( #T1_ET02 )
      wire#w1
      Contact( #O_Sal_S2 )
      I_Contact( #O_Bloqueo )
      wire#w2
      Contact( #PosTR_S2S4 )
      wire#w4
      Contact( "DB902_Estado_ZonaMesa".EstadoMesas[#Mesa].Marcha_CBx )
      I_Contact( "DB900_Estado_Mesas".EstadoVI[#Mesa].Error_Mx )
      I_Contact( "DB902_Estado_ZonaMesa".EstadoMesas[#Mesa].Manual_CBx )
      Coil( #AVTF_Sal_M2 )
   END_RUNG
   RUNG wire#powerrail
      Contact( #T1_ET10 )
   END_RUNG wire#w1
   RUNG wire#powerrail
      Contact( #T1_ET11 )
   END_RUNG wire#w1
   RUNG wire#w1
      Contact( #O_Bloqueo )
      Contact( #Mx_FlujoPrin_S2 )
   END_RUNG wire#w2
   RUNG wire#powerrail
      Contact( #T1_ET02 )
      wire#w3
      Contact( #O_Vaciar )
      Contact( #Mx_FlujoPrin_S2 )
   END_RUNG wire#w2
   RUNG wire#powerrail
      Contact( #T1_ET03 )
   END_RUNG wire#w3
   RUNG wire#powerrail
      Contact( #T1_ET60 )
   END_RUNG wire#w2
   RUNG wire#w2
      Contact( "ON" )
   END_RUNG wire#w4
   // the same network as SCL:
   #AVTF_Sal_M2 := (((#T1_ET02 OR #T1_ET10 OR #T1_ET11) AND ((#O_Sal_S2 AND NOT #O_Bloqueo) OR (#O_Bloqueo AND #Mx_FlujoPrin_S2))) OR ((#T1_ET02 OR #T1_ET03) AND #O_Vaciar AND #Mx_FlujoPrin_S2) OR #T1_ET60) AND (#PosTR_S2S4 OR "ON") AND "DB902_Estado_ZonaMesa".EstadoMesas[#Mesa].Marcha_CBx AND NOT "DB900_Estado_Mesas".EstadoVI[#Mesa].Error_Mx AND NOT "DB902_Estado_ZonaMesa".EstadoMesas[#Mesa].Manual_CBx;
END_REGION

REGION Network 42: NXT AVISO S4
   // Pablo. Damos el aviso cuando empezamos a realizar el movimiento del transfer para salir por S2
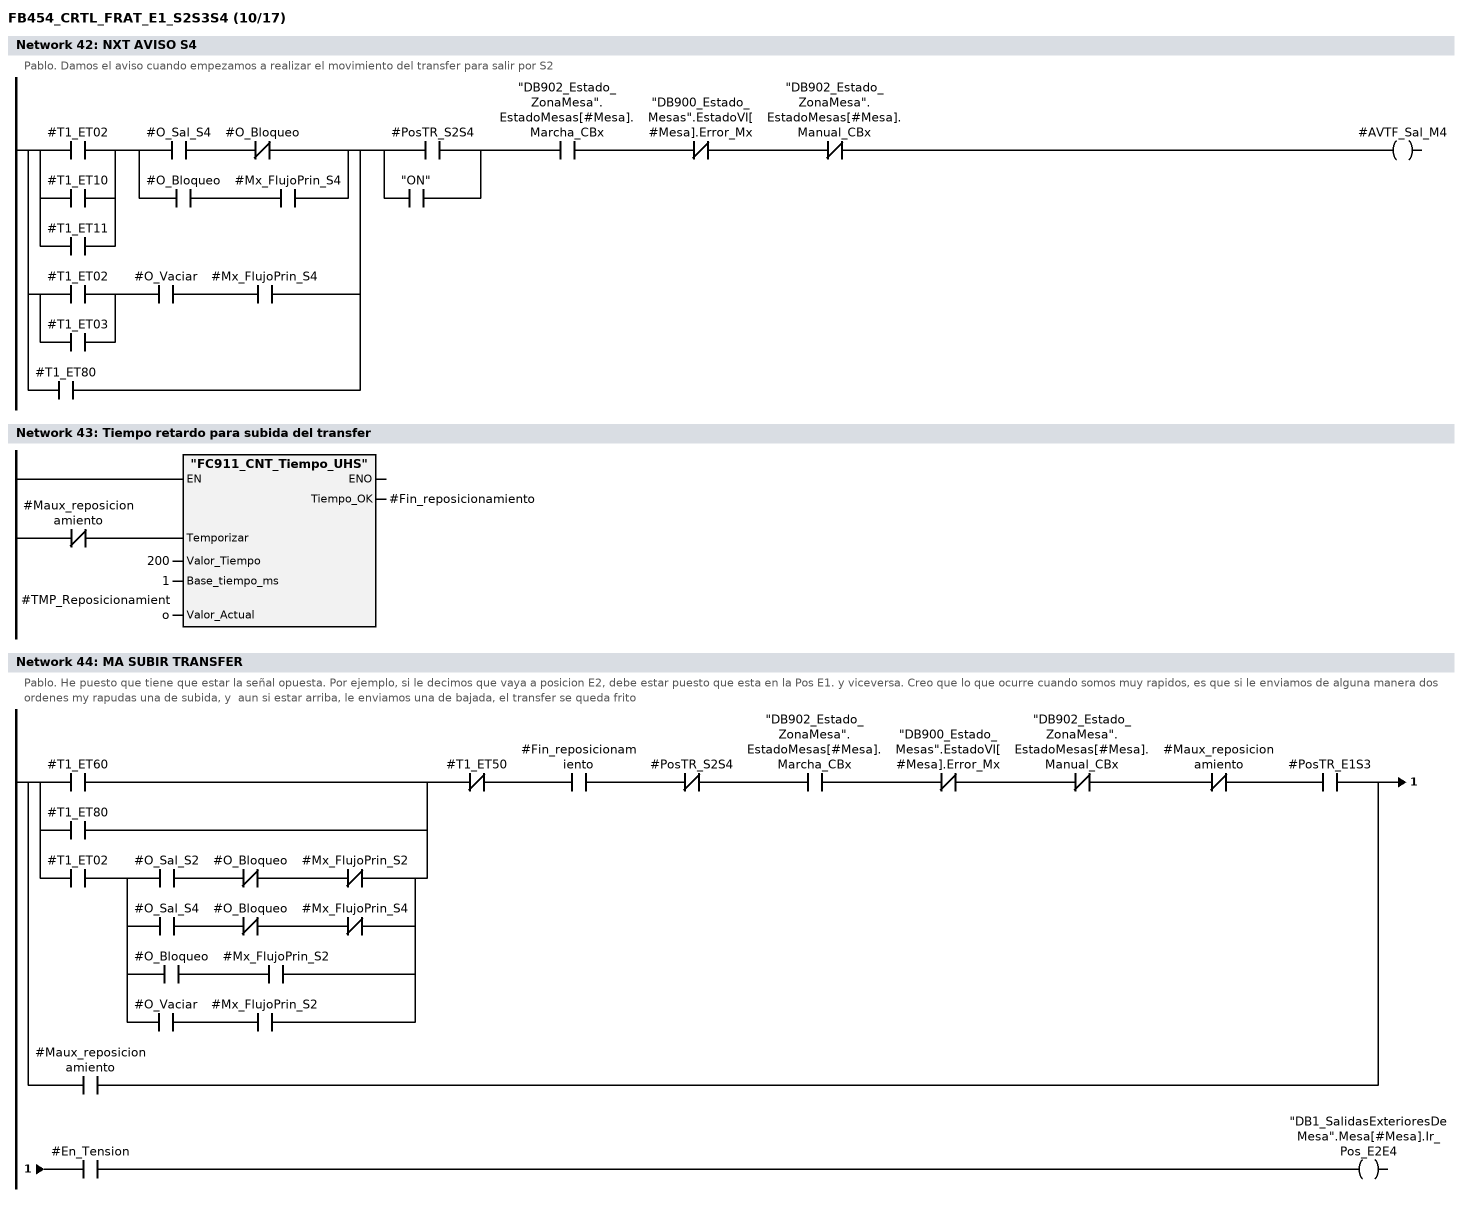
   RUNG wire#powerrail
      Contact( #T1_ET02 )
      wire#w1
      Contact( #O_Sal_S4 )
      I_Contact( #O_Bloqueo )
      wire#w2
      Contact( #PosTR_S2S4 )
      wire#w4
      Contact( "DB902_Estado_ZonaMesa".EstadoMesas[#Mesa].Marcha_CBx )
      I_Contact( "DB900_Estado_Mesas".EstadoVI[#Mesa].Error_Mx )
      I_Contact( "DB902_Estado_ZonaMesa".EstadoMesas[#Mesa].Manual_CBx )
      Coil( #AVTF_Sal_M4 )
   END_RUNG
   RUNG wire#powerrail
      Contact( #T1_ET10 )
   END_RUNG wire#w1
   RUNG wire#powerrail
      Contact( #T1_ET11 )
   END_RUNG wire#w1
   RUNG wire#w1
      Contact( #O_Bloqueo )
      Contact( #Mx_FlujoPrin_S4 )
   END_RUNG wire#w2
   RUNG wire#powerrail
      Contact( #T1_ET02 )
      wire#w3
      Contact( #O_Vaciar )
      Contact( #Mx_FlujoPrin_S4 )
   END_RUNG wire#w2
   RUNG wire#powerrail
      Contact( #T1_ET03 )
   END_RUNG wire#w3
   RUNG wire#powerrail
      Contact( #T1_ET80 )
   END_RUNG wire#w2
   RUNG wire#w2
      Contact( "ON" )
   END_RUNG wire#w4
   // the same network as SCL:
   #AVTF_Sal_M4 := (((#T1_ET02 OR #T1_ET10 OR #T1_ET11) AND ((#O_Sal_S4 AND NOT #O_Bloqueo) OR (#O_Bloqueo AND #Mx_FlujoPrin_S4))) OR ((#T1_ET02 OR #T1_ET03) AND #O_Vaciar AND #Mx_FlujoPrin_S4) OR #T1_ET80) AND (#PosTR_S2S4 OR "ON") AND "DB902_Estado_ZonaMesa".EstadoMesas[#Mesa].Marcha_CBx AND NOT "DB900_Estado_Mesas".EstadoVI[#Mesa].Error_Mx AND NOT "DB902_Estado_ZonaMesa".EstadoMesas[#Mesa].Manual_CBx;
END_REGION

REGION Network 43: Tiempo retardo para subida del transfer
   RUNG wire#powerrail
      "FC911_CNT_Tiempo_UHS"(Temporizar := wire#w1, Valor_Tiempo := 200, Base_tiempo_ms := 1, Valor_Actual := #TMP_Reposicionamiento, Tiempo_OK => #Fin_reposicionamiento)
   END_RUNG
   RUNG wire#powerrail
      I_Contact( #Maux_reposicionamiento )
   END_RUNG wire#w1
   // the same network as SCL:
   "FC911_CNT_Tiempo_UHS"(Temporizar := NOT #Maux_reposicionamiento,
                          Valor_Tiempo := 200,
                          Base_tiempo_ms := 1,
                          Valor_Actual := #TMP_Reposicionamiento,
                          Tiempo_OK => #Fin_reposicionamiento);
END_REGION

REGION Network 44: MA SUBIR TRANSFER
   // Pablo. He puesto que tiene que estar la señal opuesta. Por ejemplo, si le decimos que vaya a posicion E2, debe estar puesto que esta en la Pos E1. y viceversa. Creo que lo que ocurre cuando somos muy rapidos, es que si le enviamos de alguna manera dos ordenes my rapudas una de subida, y  aun si estar arriba, le enviamos una de bajada, el transfer se queda frito
   RUNG wire#powerrail
      Contact( #T1_ET60 )
      wire#w1
      I_Contact( #T1_ET50 )
      Contact( #Fin_reposicionamiento )
      I_Contact( #PosTR_S2S4 )
      Contact( "DB902_Estado_ZonaMesa".EstadoMesas[#Mesa].Marcha_CBx )
      I_Contact( "DB900_Estado_Mesas".EstadoVI[#Mesa].Error_Mx )
      I_Contact( "DB902_Estado_ZonaMesa".EstadoMesas[#Mesa].Manual_CBx )
      I_Contact( #Maux_reposicionamiento )
      Contact( #PosTR_E1S3 )
      wire#w3
      Contact( #En_Tension )
      Coil( "DB1_SalidasExterioresDeMesa".Mesa[#Mesa].Ir_Pos_E2E4 )
   END_RUNG
   RUNG wire#powerrail
      Contact( #T1_ET80 )
   END_RUNG wire#w1
   RUNG wire#powerrail
      Contact( #T1_ET02 )
      wire#w2
      Contact( #O_Sal_S2 )
      I_Contact( #O_Bloqueo )
      I_Contact( #Mx_FlujoPrin_S2 )
   END_RUNG wire#w1
   RUNG wire#w2
      Contact( #O_Sal_S4 )
      I_Contact( #O_Bloqueo )
      I_Contact( #Mx_FlujoPrin_S4 )
   END_RUNG wire#w1
   RUNG wire#w2
      Contact( #O_Bloqueo )
      Contact( #Mx_FlujoPrin_S2 )
   END_RUNG wire#w1
   RUNG wire#w2
      Contact( #O_Vaciar )
      Contact( #Mx_FlujoPrin_S2 )
   END_RUNG wire#w1
   RUNG wire#powerrail
      Contact( #Maux_reposicionamiento )
   END_RUNG wire#w3
   // the same network as SCL:
   "DB1_SalidasExterioresDeMesa".Mesa[#Mesa].Ir_Pos_E2E4 := (((#T1_ET60 OR #T1_ET80 OR (#T1_ET02 AND ((#O_Sal_S2 AND NOT #O_Bloqueo AND NOT #Mx_FlujoPrin_S2) OR (#O_Sal_S4 AND NOT #O_Bloqueo AND NOT #Mx_FlujoPrin_S4) OR (#O_Bloqueo AND #Mx_FlujoPrin_S2) OR (#O_Vaciar AND #Mx_FlujoPrin_S2)))) AND NOT #T1_ET50 AND #Fin_reposicionamiento AND NOT #PosTR_S2S4 AND "DB902_Estado_ZonaMesa".EstadoMesas[#Mesa].Marcha_CBx AND NOT "DB900_Estado_Mesas".EstadoVI[#Mesa].Error_Mx AND NOT "DB902_Estado_ZonaMesa".EstadoMesas[#Mesa].Manual_CBx AND NOT #Maux_reposicionamiento AND #PosTR_E1S3) OR #Maux_reposicionamiento) AND #En_Tension;
END_REGION

REGION Network 45: MA ir posicion 1-3
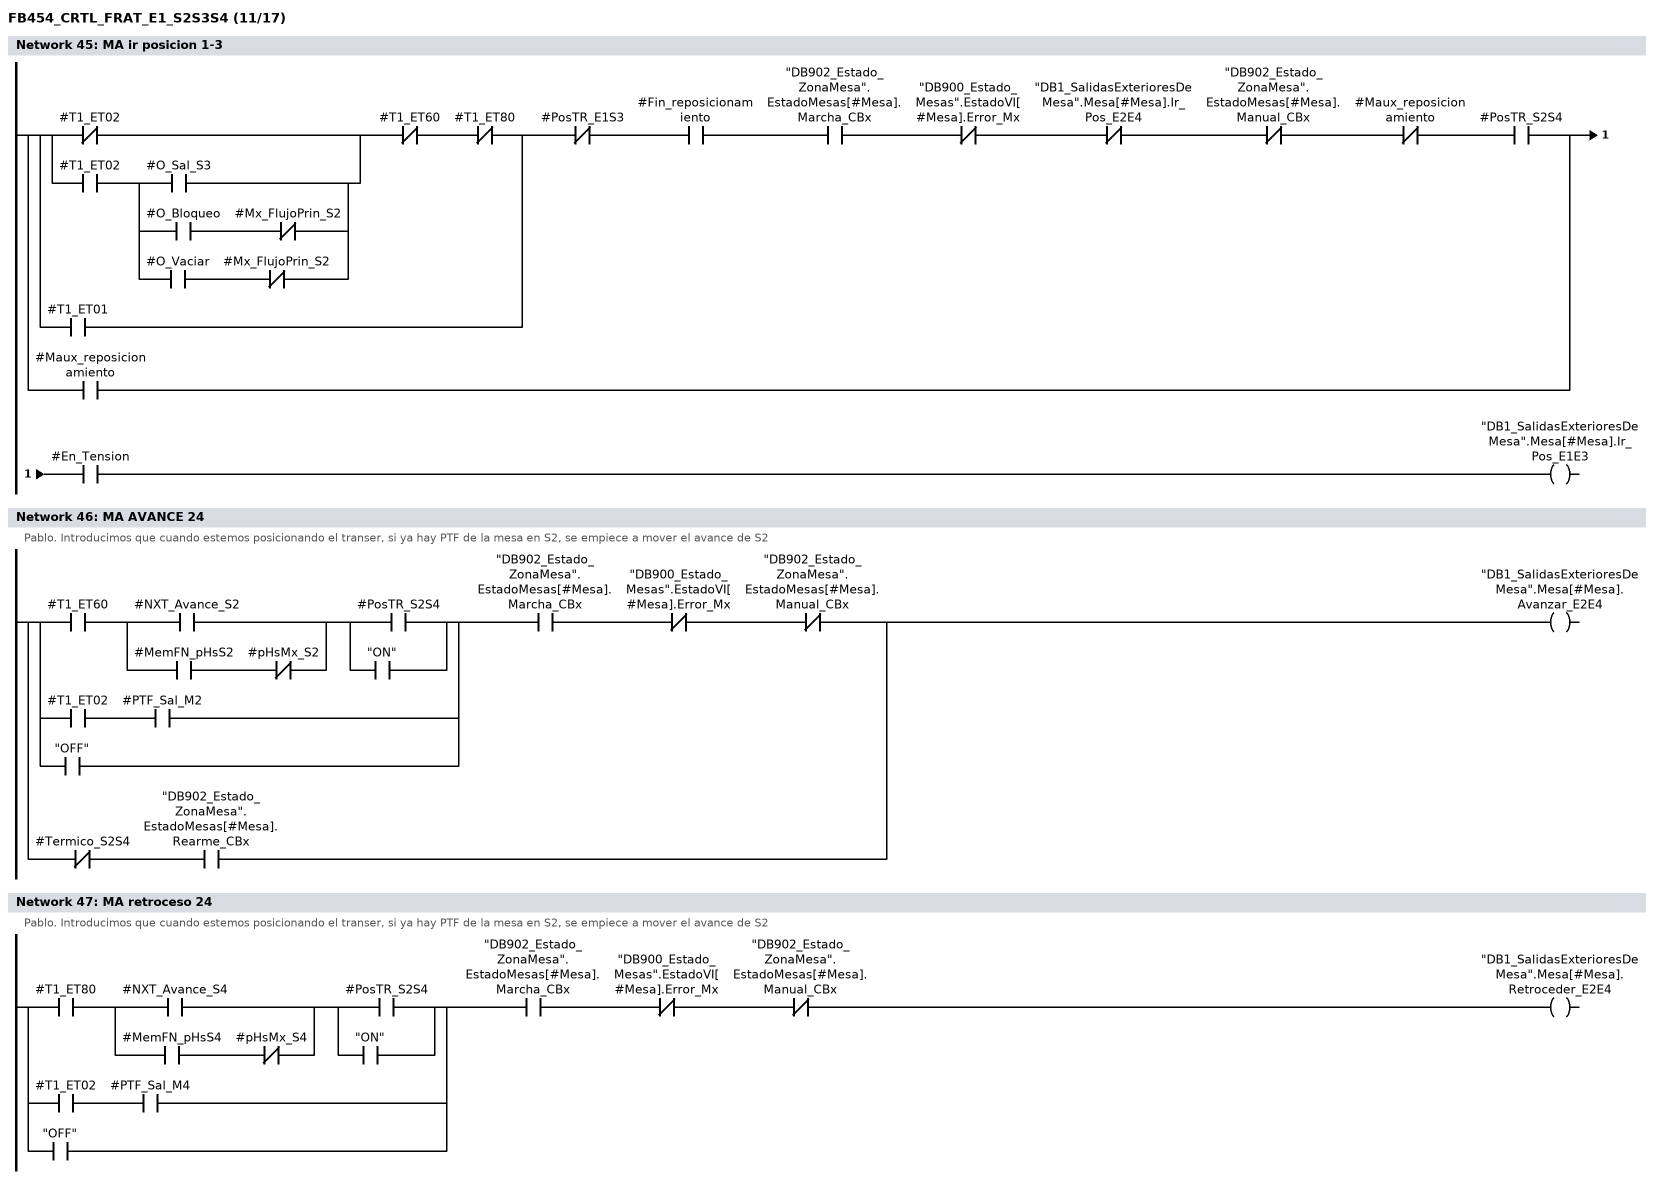
   RUNG wire#powerrail
      I_Contact( #T1_ET02 )
      wire#w1
      I_Contact( #T1_ET60 )
      I_Contact( #T1_ET80 )
      wire#w3
      I_Contact( #PosTR_E1S3 )
      Contact( #Fin_reposicionamiento )
      Contact( "DB902_Estado_ZonaMesa".EstadoMesas[#Mesa].Marcha_CBx )
      I_Contact( "DB900_Estado_Mesas".EstadoVI[#Mesa].Error_Mx )
      I_Contact( "DB1_SalidasExterioresDeMesa".Mesa[#Mesa].Ir_Pos_E2E4 )
      I_Contact( "DB902_Estado_ZonaMesa".EstadoMesas[#Mesa].Manual_CBx )
      I_Contact( #Maux_reposicionamiento )
      Contact( #PosTR_S2S4 )
      wire#w4
      Contact( #En_Tension )
      Coil( "DB1_SalidasExterioresDeMesa".Mesa[#Mesa].Ir_Pos_E1E3 )
   END_RUNG
   RUNG wire#powerrail
      Contact( #T1_ET02 )
      wire#w2
      Contact( #O_Sal_S3 )
   END_RUNG wire#w1
   RUNG wire#w2
      Contact( #O_Bloqueo )
      I_Contact( #Mx_FlujoPrin_S2 )
   END_RUNG wire#w1
   RUNG wire#w2
      Contact( #O_Vaciar )
      I_Contact( #Mx_FlujoPrin_S2 )
   END_RUNG wire#w1
   RUNG wire#powerrail
      Contact( #T1_ET01 )
   END_RUNG wire#w3
   RUNG wire#powerrail
      Contact( #Maux_reposicionamiento )
   END_RUNG wire#w4
   // the same network as SCL:
   "DB1_SalidasExterioresDeMesa".Mesa[#Mesa].Ir_Pos_E1E3 := (((((NOT #T1_ET02 OR (#T1_ET02 AND (#O_Sal_S3 OR (#O_Bloqueo AND NOT #Mx_FlujoPrin_S2) OR (#O_Vaciar AND NOT #Mx_FlujoPrin_S2)))) AND NOT #T1_ET60 AND NOT #T1_ET80) OR #T1_ET01) AND NOT #PosTR_E1S3 AND #Fin_reposicionamiento AND "DB902_Estado_ZonaMesa".EstadoMesas[#Mesa].Marcha_CBx AND NOT "DB900_Estado_Mesas".EstadoVI[#Mesa].Error_Mx AND NOT "DB1_SalidasExterioresDeMesa".Mesa[#Mesa].Ir_Pos_E2E4 AND NOT "DB902_Estado_ZonaMesa".EstadoMesas[#Mesa].Manual_CBx AND NOT #Maux_reposicionamiento AND #PosTR_S2S4) OR #Maux_reposicionamiento) AND #En_Tension;
END_REGION

REGION Network 46: MA AVANCE 24
   // Pablo. Introducimos que cuando estemos posicionando el transer, si ya hay PTF de la mesa en S2, se empiece a mover el avance de S2
   RUNG wire#powerrail
      Contact( #T1_ET60 )
      wire#w1
      Contact( #NXT_Avance_S2 )
      wire#w2
      Contact( #PosTR_S2S4 )
      wire#w3
      Contact( "DB902_Estado_ZonaMesa".EstadoMesas[#Mesa].Marcha_CBx )
      I_Contact( "DB900_Estado_Mesas".EstadoVI[#Mesa].Error_Mx )
      I_Contact( "DB902_Estado_ZonaMesa".EstadoMesas[#Mesa].Manual_CBx )
      wire#w4
      Coil( "DB1_SalidasExterioresDeMesa".Mesa[#Mesa].Avanzar_E2E4 )
   END_RUNG
   RUNG wire#w1
      Contact( #MemFN_pHsS2 )
      I_Contact( #pHsMx_S2 )
   END_RUNG wire#w2
   RUNG wire#w2
      Contact( "ON" )
   END_RUNG wire#w3
   RUNG wire#powerrail
      Contact( #T1_ET02 )
      Contact( #PTF_Sal_M2 )
   END_RUNG wire#w3
   RUNG wire#powerrail
      Contact( "OFF" )
   END_RUNG wire#w3
   RUNG wire#powerrail
      I_Contact( #Termico_S2S4 )
      Contact( "DB902_Estado_ZonaMesa".EstadoMesas[#Mesa].Rearme_CBx )
   END_RUNG wire#w4
   // the same network as SCL:
   "DB1_SalidasExterioresDeMesa".Mesa[#Mesa].Avanzar_E2E4 := (((#T1_ET60 AND (#NXT_Avance_S2 OR (#MemFN_pHsS2 AND NOT #pHsMx_S2)) AND (#PosTR_S2S4 OR "ON")) OR (#T1_ET02 AND #PTF_Sal_M2) OR "OFF") AND "DB902_Estado_ZonaMesa".EstadoMesas[#Mesa].Marcha_CBx AND NOT "DB900_Estado_Mesas".EstadoVI[#Mesa].Error_Mx AND NOT "DB902_Estado_ZonaMesa".EstadoMesas[#Mesa].Manual_CBx) OR (NOT #Termico_S2S4 AND "DB902_Estado_ZonaMesa".EstadoMesas[#Mesa].Rearme_CBx);
END_REGION

REGION Network 47: MA retroceso 24
   // Pablo. Introducimos que cuando estemos posicionando el transer, si ya hay PTF de la mesa en S2, se empiece a mover el avance de S2
   RUNG wire#powerrail
      Contact( #T1_ET80 )
      wire#w1
      Contact( #NXT_Avance_S4 )
      wire#w2
      Contact( #PosTR_S2S4 )
      wire#w3
      Contact( "DB902_Estado_ZonaMesa".EstadoMesas[#Mesa].Marcha_CBx )
      I_Contact( "DB900_Estado_Mesas".EstadoVI[#Mesa].Error_Mx )
      I_Contact( "DB902_Estado_ZonaMesa".EstadoMesas[#Mesa].Manual_CBx )
      Coil( "DB1_SalidasExterioresDeMesa".Mesa[#Mesa].Retroceder_E2E4 )
   END_RUNG
   RUNG wire#w1
      Contact( #MemFN_pHsS4 )
      I_Contact( #pHsMx_S4 )
   END_RUNG wire#w2
   RUNG wire#w2
      Contact( "ON" )
   END_RUNG wire#w3
   RUNG wire#powerrail
      Contact( #T1_ET02 )
      Contact( #PTF_Sal_M4 )
   END_RUNG wire#w3
   RUNG wire#powerrail
      Contact( "OFF" )
   END_RUNG wire#w3
   // the same network as SCL:
   "DB1_SalidasExterioresDeMesa".Mesa[#Mesa].Retroceder_E2E4 := ((#T1_ET80 AND (#NXT_Avance_S4 OR (#MemFN_pHsS4 AND NOT #pHsMx_S4)) AND (#PosTR_S2S4 OR "ON")) OR (#T1_ET02 AND #PTF_Sal_M4) OR "OFF") AND "DB902_Estado_ZonaMesa".EstadoMesas[#Mesa].Marcha_CBx AND NOT "DB900_Estado_Mesas".EstadoVI[#Mesa].Error_Mx AND NOT "DB902_Estado_ZonaMesa".EstadoMesas[#Mesa].Manual_CBx;
END_REGION

REGION Network 48: Memoria, Para optimizar el movimiento del Motor E1 y no avanzar mas de la cuenta
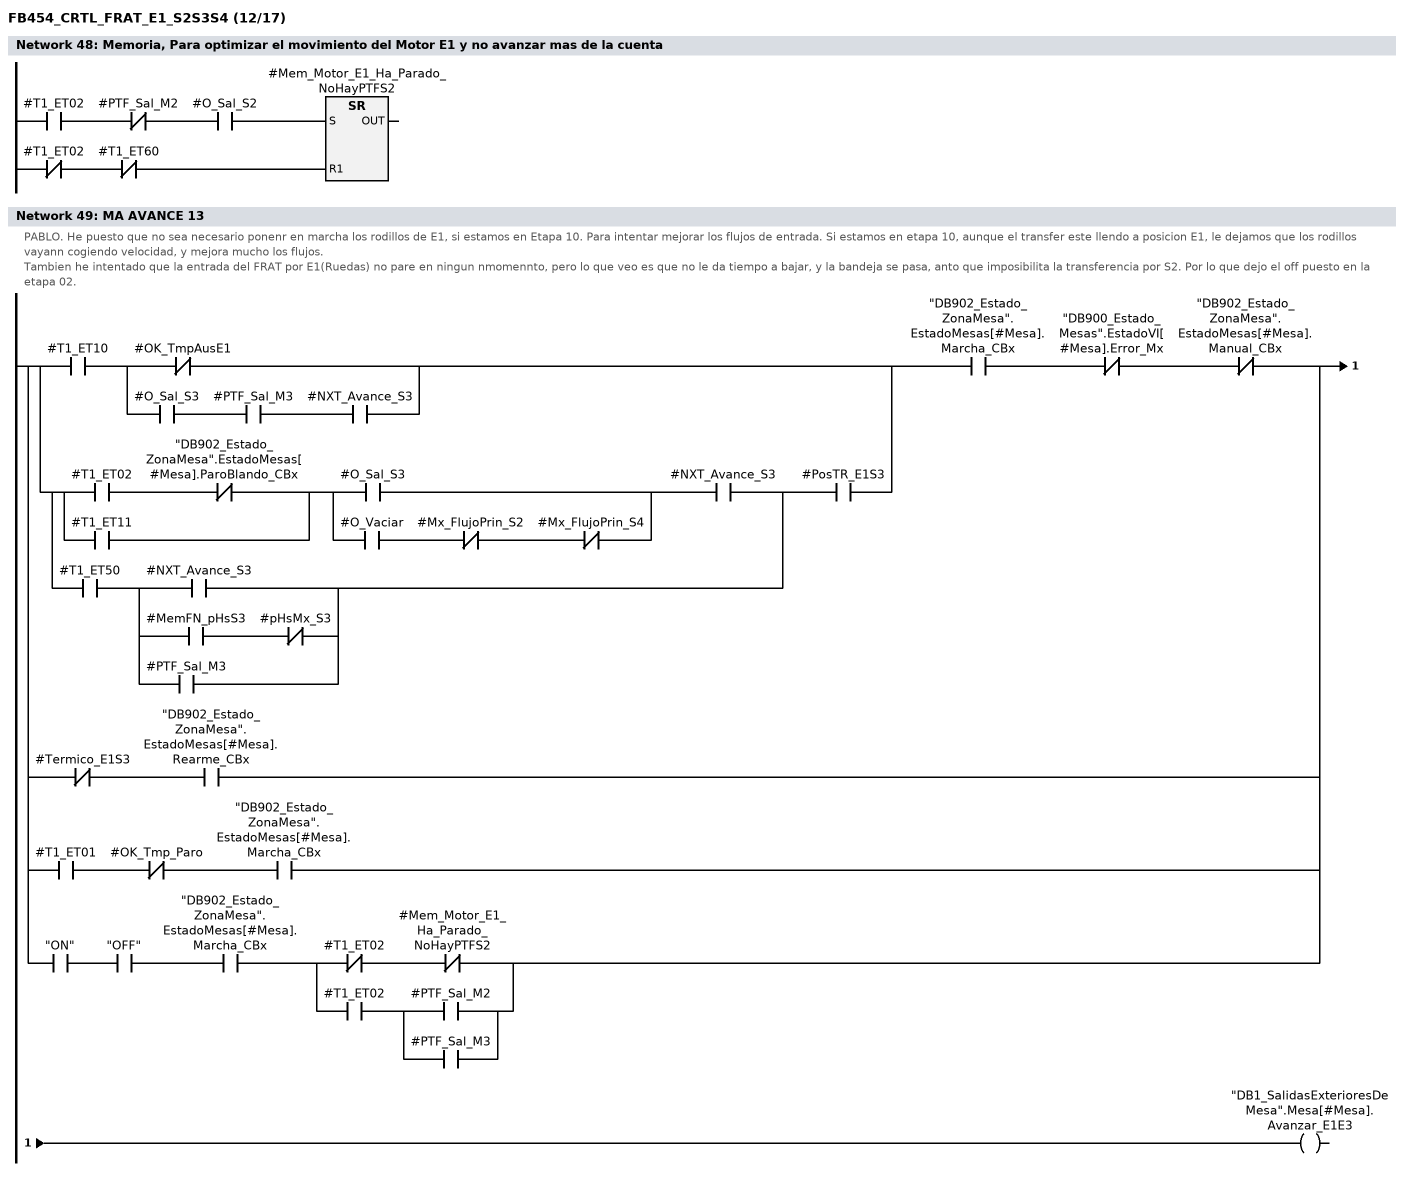
   RUNG wire#powerrail
      Contact( #T1_ET02 )
      I_Contact( #PTF_Sal_M2 )
      Contact( #O_Sal_S2 )
      S_SR(operand := #Mem_Motor_E1_Ha_Parado_NoHayPTFS2, r1 := wire#w1)
   END_RUNG
   RUNG wire#powerrail
      I_Contact( #T1_ET02 )
      I_Contact( #T1_ET60 )
   END_RUNG wire#w1
   // the same network as SCL:
   IF #T1_ET02 AND NOT #PTF_Sal_M2 AND #O_Sal_S2 THEN
       #Mem_Motor_E1_Ha_Parado_NoHayPTFS2 := TRUE;   // SR flip-flop
   END_IF;
   IF NOT #T1_ET02 AND NOT #T1_ET60 THEN #Mem_Motor_E1_Ha_Parado_NoHayPTFS2 := FALSE; END_IF;
END_REGION

REGION Network 49: MA AVANCE 13
   // PABLO. He puesto que no sea necesario ponenr en marcha los rodillos de E1, si estamos en Etapa 10. Para intentar mejorar los flujos de entrada. Si estamos en etapa 10, aunque el transfer este llendo a posicion E1, le dejamos que los rodillos vayann cogiendo velocidad, y mejora mucho los flujos. 
   // Tambien he intentado que la entrada del FRAT por E1(Ruedas) no pare en ningun nmomennto, pero lo que veo es que no le da tiempo a bajar, y la bandeja se pasa, anto que imposibilita la transferencia por S2. Por lo que dejo el off puesto en la etapa 02.
   RUNG wire#powerrail
      Contact( #T1_ET10 )
      wire#w1
      I_Contact( #OK_TmpAusE1 )
      wire#w2
      Contact( "DB902_Estado_ZonaMesa".EstadoMesas[#Mesa].Marcha_CBx )
      I_Contact( "DB900_Estado_Mesas".EstadoVI[#Mesa].Error_Mx )
      I_Contact( "DB902_Estado_ZonaMesa".EstadoMesas[#Mesa].Manual_CBx )
      wire#w7
      Coil( "DB1_SalidasExterioresDeMesa".Mesa[#Mesa].Avanzar_E1E3 )
   END_RUNG
   RUNG wire#w1
      Contact( #O_Sal_S3 )
      Contact( #PTF_Sal_M3 )
      Contact( #NXT_Avance_S3 )
   END_RUNG wire#w2
   RUNG wire#powerrail
      Contact( #T1_ET02 )
      I_Contact( "DB902_Estado_ZonaMesa".EstadoMesas[#Mesa].ParoBlando_CBx )
      wire#w3
      Contact( #O_Sal_S3 )
      wire#w4
      Contact( #NXT_Avance_S3 )
      wire#w5
      Contact( #PosTR_E1S3 )
   END_RUNG wire#w2
   RUNG wire#powerrail
      Contact( #T1_ET11 )
   END_RUNG wire#w3
   RUNG wire#w3
      Contact( #O_Vaciar )
      I_Contact( #Mx_FlujoPrin_S2 )
      I_Contact( #Mx_FlujoPrin_S4 )
   END_RUNG wire#w4
   RUNG wire#powerrail
      Contact( #T1_ET50 )
      wire#w6
      Contact( #NXT_Avance_S3 )
   END_RUNG wire#w5
   RUNG wire#w6
      Contact( #MemFN_pHsS3 )
      I_Contact( #pHsMx_S3 )
   END_RUNG wire#w5
   RUNG wire#w6
      Contact( #PTF_Sal_M3 )
   END_RUNG wire#w5
   RUNG wire#powerrail
      I_Contact( #Termico_E1S3 )
      Contact( "DB902_Estado_ZonaMesa".EstadoMesas[#Mesa].Rearme_CBx )
   END_RUNG wire#w7
   RUNG wire#powerrail
      Contact( #T1_ET01 )
      I_Contact( #OK_Tmp_Paro )
      Contact( "DB902_Estado_ZonaMesa".EstadoMesas[#Mesa].Marcha_CBx )
   END_RUNG wire#w7
   RUNG wire#powerrail
      Contact( "ON" )
      Contact( "OFF" )
      Contact( "DB902_Estado_ZonaMesa".EstadoMesas[#Mesa].Marcha_CBx )
      wire#w8
      I_Contact( #T1_ET02 )
      I_Contact( #Mem_Motor_E1_Ha_Parado_NoHayPTFS2 )
   END_RUNG wire#w7
   RUNG wire#w8
      Contact( #T1_ET02 )
      wire#w9
      Contact( #PTF_Sal_M2 )
   END_RUNG wire#w7
   RUNG wire#w9
      Contact( #PTF_Sal_M3 )
   END_RUNG wire#w7
   // the same network as SCL:
   "DB1_SalidasExterioresDeMesa".Mesa[#Mesa].Avanzar_E1E3 := (((#T1_ET10 AND (NOT #OK_TmpAusE1 OR (#O_Sal_S3 AND #PTF_Sal_M3 AND #NXT_Avance_S3))) OR (((((#T1_ET02 AND NOT "DB902_Estado_ZonaMesa".EstadoMesas[#Mesa].ParoBlando_CBx) OR #T1_ET11) AND (#O_Sal_S3 OR (#O_Vaciar AND NOT #Mx_FlujoPrin_S2 AND NOT #Mx_FlujoPrin_S4)) AND #NXT_Avance_S3) OR (#T1_ET50 AND (#NXT_Avance_S3 OR (#MemFN_pHsS3 AND NOT #pHsMx_S3) OR #PTF_Sal_M3))) AND #PosTR_E1S3)) AND "DB902_Estado_ZonaMesa".EstadoMesas[#Mesa].Marcha_CBx AND NOT "DB900_Estado_Mesas".EstadoVI[#Mesa].Error_Mx AND NOT "DB902_Estado_ZonaMesa".EstadoMesas[#Mesa].Manual_CBx) OR (NOT #Termico_E1S3 AND "DB902_Estado_ZonaMesa".EstadoMesas[#Mesa].Rearme_CBx) OR (#T1_ET01 AND NOT #OK_Tmp_Paro AND "DB902_Estado_ZonaMesa".EstadoMesas[#Mesa].Marcha_CBx) OR ("ON" AND "OFF" AND "DB902_Estado_ZonaMesa".EstadoMesas[#Mesa].Marcha_CBx AND ((NOT #T1_ET02 AND NOT #Mem_Motor_E1_Ha_Parado_NoHayPTFS2) OR (#T1_ET02 AND (#PTF_Sal_M2 OR #PTF_Sal_M3))));
END_REGION

REGION Network 50: PASAR ETIQUETA JDT
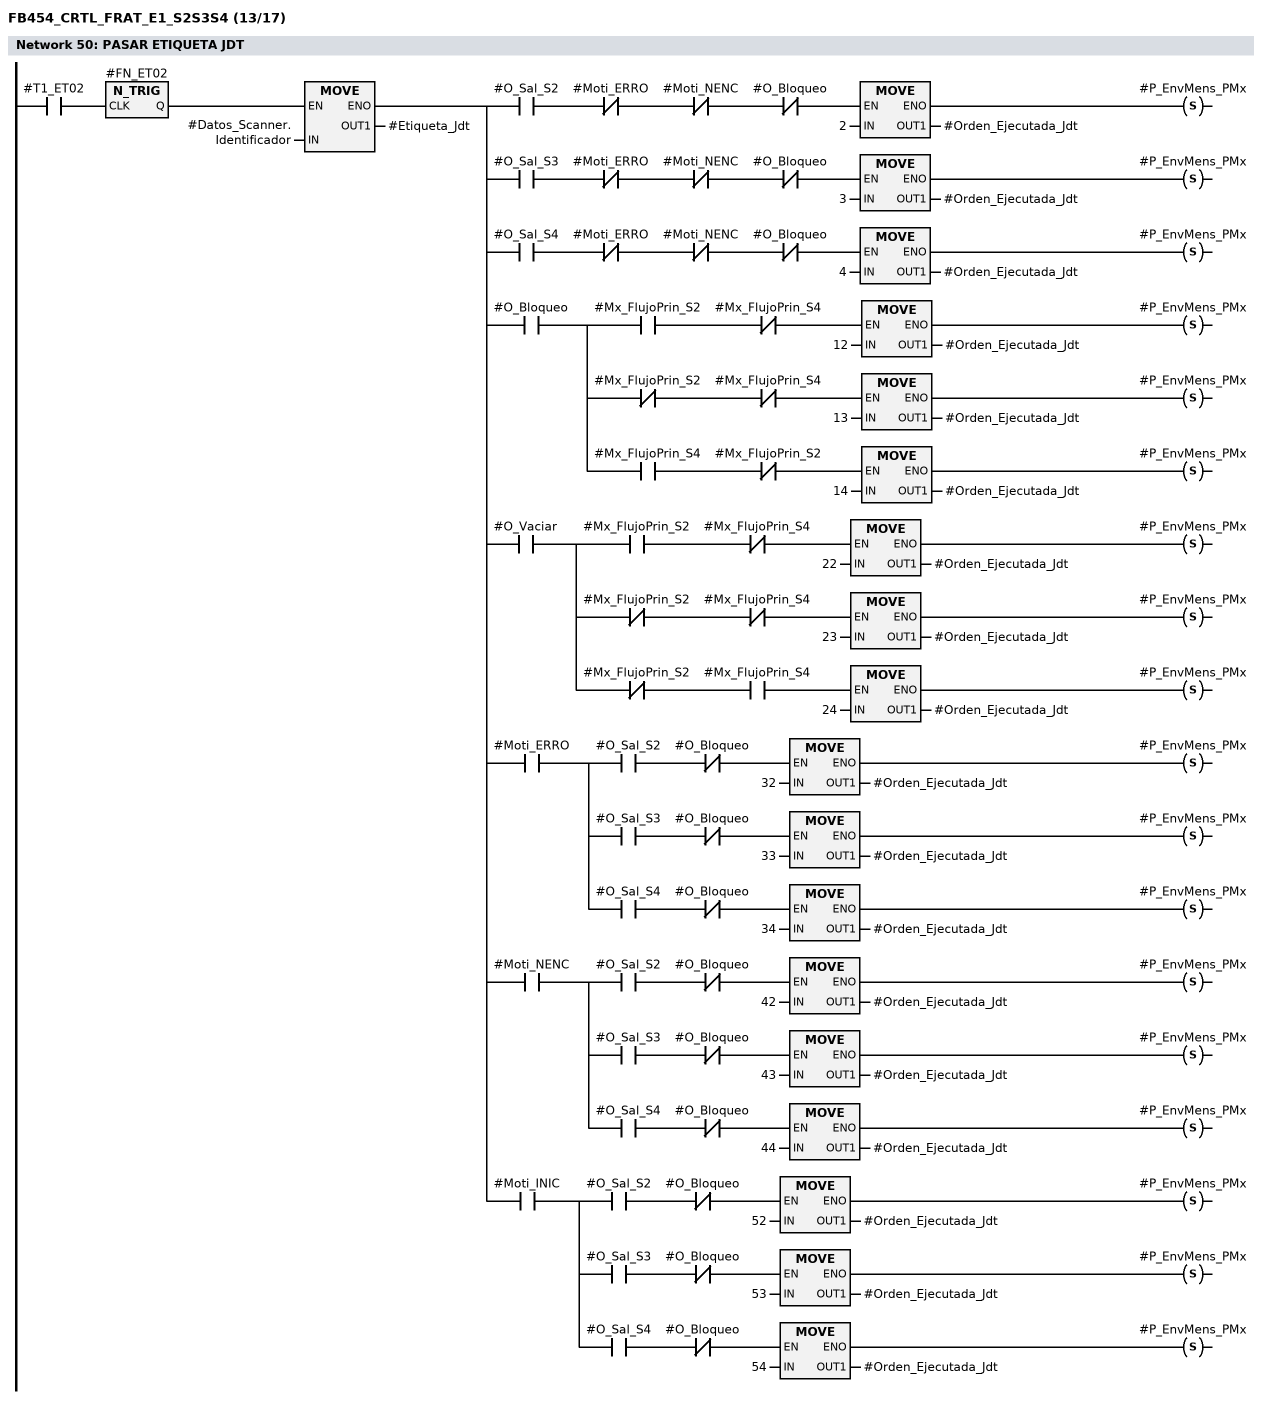
   RUNG wire#powerrail
      Contact( #T1_ET02 )
      N_Trig( #FN_ET02 )
      { S7_GenerateENO := "TRUE" } Move(in := #Datos_Scanner.Identificador, out1 => #Etiqueta_Jdt)
      wire#w1
      Contact( #O_Sal_S2 )
      I_Contact( #Moti_ERRO )
      I_Contact( #Moti_NENC )
      I_Contact( #O_Bloqueo )
      { S7_GenerateENO := "TRUE" } Move(in := 2, out1 => #Orden_Ejecutada_Jdt)
      S_Coil( #P_EnvMens_PMx )
   END_RUNG
   RUNG wire#w1
      Contact( #O_Sal_S3 )
      I_Contact( #Moti_ERRO )
      I_Contact( #Moti_NENC )
      I_Contact( #O_Bloqueo )
      { S7_GenerateENO := "TRUE" } Move(in := 3, out1 => #Orden_Ejecutada_Jdt)
      S_Coil( #P_EnvMens_PMx )
   END_RUNG
   RUNG wire#w1
      Contact( #O_Sal_S4 )
      I_Contact( #Moti_ERRO )
      I_Contact( #Moti_NENC )
      I_Contact( #O_Bloqueo )
      { S7_GenerateENO := "TRUE" } Move(in := 4, out1 => #Orden_Ejecutada_Jdt)
      S_Coil( #P_EnvMens_PMx )
   END_RUNG
   RUNG wire#w1
      Contact( #O_Bloqueo )
      wire#w2
      Contact( #Mx_FlujoPrin_S2 )
      I_Contact( #Mx_FlujoPrin_S4 )
      { S7_GenerateENO := "TRUE" } Move(in := 12, out1 => #Orden_Ejecutada_Jdt)
      S_Coil( #P_EnvMens_PMx )
   END_RUNG
   RUNG wire#w2
      I_Contact( #Mx_FlujoPrin_S2 )
      I_Contact( #Mx_FlujoPrin_S4 )
      { S7_GenerateENO := "TRUE" } Move(in := 13, out1 => #Orden_Ejecutada_Jdt)
      S_Coil( #P_EnvMens_PMx )
   END_RUNG
   RUNG wire#w2
      Contact( #Mx_FlujoPrin_S4 )
      I_Contact( #Mx_FlujoPrin_S2 )
      { S7_GenerateENO := "TRUE" } Move(in := 14, out1 => #Orden_Ejecutada_Jdt)
      S_Coil( #P_EnvMens_PMx )
   END_RUNG
   RUNG wire#w1
      Contact( #O_Vaciar )
      wire#w3
      Contact( #Mx_FlujoPrin_S2 )
      I_Contact( #Mx_FlujoPrin_S4 )
      { S7_GenerateENO := "TRUE" } Move(in := 22, out1 => #Orden_Ejecutada_Jdt)
      S_Coil( #P_EnvMens_PMx )
   END_RUNG
   RUNG wire#w3
      I_Contact( #Mx_FlujoPrin_S2 )
      I_Contact( #Mx_FlujoPrin_S4 )
      { S7_GenerateENO := "TRUE" } Move(in := 23, out1 => #Orden_Ejecutada_Jdt)
      S_Coil( #P_EnvMens_PMx )
   END_RUNG
   RUNG wire#w3
      I_Contact( #Mx_FlujoPrin_S2 )
      Contact( #Mx_FlujoPrin_S4 )
      { S7_GenerateENO := "TRUE" } Move(in := 24, out1 => #Orden_Ejecutada_Jdt)
      S_Coil( #P_EnvMens_PMx )
   END_RUNG
   RUNG wire#w1
      Contact( #Moti_ERRO )
      wire#w4
      Contact( #O_Sal_S2 )
      I_Contact( #O_Bloqueo )
      { S7_GenerateENO := "TRUE" } Move(in := 32, out1 => #Orden_Ejecutada_Jdt)
      S_Coil( #P_EnvMens_PMx )
   END_RUNG
   RUNG wire#w4
      Contact( #O_Sal_S3 )
      I_Contact( #O_Bloqueo )
      { S7_GenerateENO := "TRUE" } Move(in := 33, out1 => #Orden_Ejecutada_Jdt)
      S_Coil( #P_EnvMens_PMx )
   END_RUNG
   RUNG wire#w4
      Contact( #O_Sal_S4 )
      I_Contact( #O_Bloqueo )
      { S7_GenerateENO := "TRUE" } Move(in := 34, out1 => #Orden_Ejecutada_Jdt)
      S_Coil( #P_EnvMens_PMx )
   END_RUNG
   RUNG wire#w1
      Contact( #Moti_NENC )
      wire#w5
      Contact( #O_Sal_S2 )
      I_Contact( #O_Bloqueo )
      { S7_GenerateENO := "TRUE" } Move(in := 42, out1 => #Orden_Ejecutada_Jdt)
      S_Coil( #P_EnvMens_PMx )
   END_RUNG
   RUNG wire#w5
      Contact( #O_Sal_S3 )
      I_Contact( #O_Bloqueo )
      { S7_GenerateENO := "TRUE" } Move(in := 43, out1 => #Orden_Ejecutada_Jdt)
      S_Coil( #P_EnvMens_PMx )
   END_RUNG
   RUNG wire#w5
      Contact( #O_Sal_S4 )
      I_Contact( #O_Bloqueo )
      { S7_GenerateENO := "TRUE" } Move(in := 44, out1 => #Orden_Ejecutada_Jdt)
      S_Coil( #P_EnvMens_PMx )
   END_RUNG
   RUNG wire#w1
      Contact( #Moti_INIC )
      wire#w6
      Contact( #O_Sal_S2 )
      I_Contact( #O_Bloqueo )
      { S7_GenerateENO := "TRUE" } Move(in := 52, out1 => #Orden_Ejecutada_Jdt)
      S_Coil( #P_EnvMens_PMx )
   END_RUNG
   RUNG wire#w6
      Contact( #O_Sal_S3 )
      I_Contact( #O_Bloqueo )
      { S7_GenerateENO := "TRUE" } Move(in := 53, out1 => #Orden_Ejecutada_Jdt)
      S_Coil( #P_EnvMens_PMx )
   END_RUNG
   RUNG wire#w6
      Contact( #O_Sal_S4 )
      I_Contact( #O_Bloqueo )
      { S7_GenerateENO := "TRUE" } Move(in := 54, out1 => #Orden_Ejecutada_Jdt)
      S_Coil( #P_EnvMens_PMx )
   END_RUNG
   // the same network as SCL:
   // ENO of a box is taken as its EN; it also drops when the box reports an error
   #_w1 := NOT #T1_ET02 AND #FN_ET02;   // falling edge
   #FN_ET02 := #T1_ET02;
   IF #_w1 THEN #Etiqueta_Jdt := #Datos_Scanner.Identificador; END_IF;
   IF #_w1 AND #O_Sal_S2 AND NOT #Moti_ERRO AND NOT #Moti_NENC AND NOT #O_Bloqueo THEN
       #Orden_Ejecutada_Jdt := 2;
       #P_EnvMens_PMx := TRUE;
   END_IF;
   IF #_w1 AND #O_Sal_S3 AND NOT #Moti_ERRO AND NOT #Moti_NENC AND NOT #O_Bloqueo THEN
       #Orden_Ejecutada_Jdt := 3;
       #P_EnvMens_PMx := TRUE;
   END_IF;
   IF #_w1 AND #O_Sal_S4 AND NOT #Moti_ERRO AND NOT #Moti_NENC AND NOT #O_Bloqueo THEN
       #Orden_Ejecutada_Jdt := 4;
       #P_EnvMens_PMx := TRUE;
   END_IF;
   #_w2 := #_w1 AND #O_Bloqueo;
   IF #_w2 AND #Mx_FlujoPrin_S2 AND NOT #Mx_FlujoPrin_S4 THEN
       #Orden_Ejecutada_Jdt := 12;
       #P_EnvMens_PMx := TRUE;
   END_IF;
   IF #_w2 AND NOT #Mx_FlujoPrin_S2 AND NOT #Mx_FlujoPrin_S4 THEN
       #Orden_Ejecutada_Jdt := 13;
       #P_EnvMens_PMx := TRUE;
   END_IF;
   IF #_w2 AND #Mx_FlujoPrin_S4 AND NOT #Mx_FlujoPrin_S2 THEN
       #Orden_Ejecutada_Jdt := 14;
       #P_EnvMens_PMx := TRUE;
   END_IF;
   #_w3 := #_w1 AND #O_Vaciar;
   IF #_w3 AND #Mx_FlujoPrin_S2 AND NOT #Mx_FlujoPrin_S4 THEN
       #Orden_Ejecutada_Jdt := 22;
       #P_EnvMens_PMx := TRUE;
   END_IF;
   IF #_w3 AND NOT #Mx_FlujoPrin_S2 AND NOT #Mx_FlujoPrin_S4 THEN
       #Orden_Ejecutada_Jdt := 23;
       #P_EnvMens_PMx := TRUE;
   END_IF;
   IF #_w3 AND NOT #Mx_FlujoPrin_S2 AND #Mx_FlujoPrin_S4 THEN
       #Orden_Ejecutada_Jdt := 24;
       #P_EnvMens_PMx := TRUE;
   END_IF;
   #_w4 := #_w1 AND #Moti_ERRO;
   IF #_w4 AND #O_Sal_S2 AND NOT #O_Bloqueo THEN
       #Orden_Ejecutada_Jdt := 32;
       #P_EnvMens_PMx := TRUE;
   END_IF;
   IF #_w4 AND #O_Sal_S3 AND NOT #O_Bloqueo THEN
       #Orden_Ejecutada_Jdt := 33;
       #P_EnvMens_PMx := TRUE;
   END_IF;
   IF #_w4 AND #O_Sal_S4 AND NOT #O_Bloqueo THEN
       #Orden_Ejecutada_Jdt := 34;
       #P_EnvMens_PMx := TRUE;
   END_IF;
   #_w5 := #_w1 AND #Moti_NENC;
   IF #_w5 AND #O_Sal_S2 AND NOT #O_Bloqueo THEN
       #Orden_Ejecutada_Jdt := 42;
       #P_EnvMens_PMx := TRUE;
   END_IF;
   IF #_w5 AND #O_Sal_S3 AND NOT #O_Bloqueo THEN
       #Orden_Ejecutada_Jdt := 43;
       #P_EnvMens_PMx := TRUE;
   END_IF;
   IF #_w5 AND #O_Sal_S4 AND NOT #O_Bloqueo THEN
       #Orden_Ejecutada_Jdt := 44;
       #P_EnvMens_PMx := TRUE;
   END_IF;
   #_w6 := #_w1 AND #Moti_INIC;
   IF #_w6 AND #O_Sal_S2 AND NOT #O_Bloqueo THEN
       #Orden_Ejecutada_Jdt := 52;
       #P_EnvMens_PMx := TRUE;
   END_IF;
   IF #_w6 AND #O_Sal_S3 AND NOT #O_Bloqueo THEN
       #Orden_Ejecutada_Jdt := 53;
       #P_EnvMens_PMx := TRUE;
   END_IF;
   IF #_w6 AND #O_Sal_S4 AND NOT #O_Bloqueo THEN
       #Orden_Ejecutada_Jdt := 54;
       #P_EnvMens_PMx := TRUE;
   END_IF;
END_REGION

REGION Network 51: RESET PRESENCIA
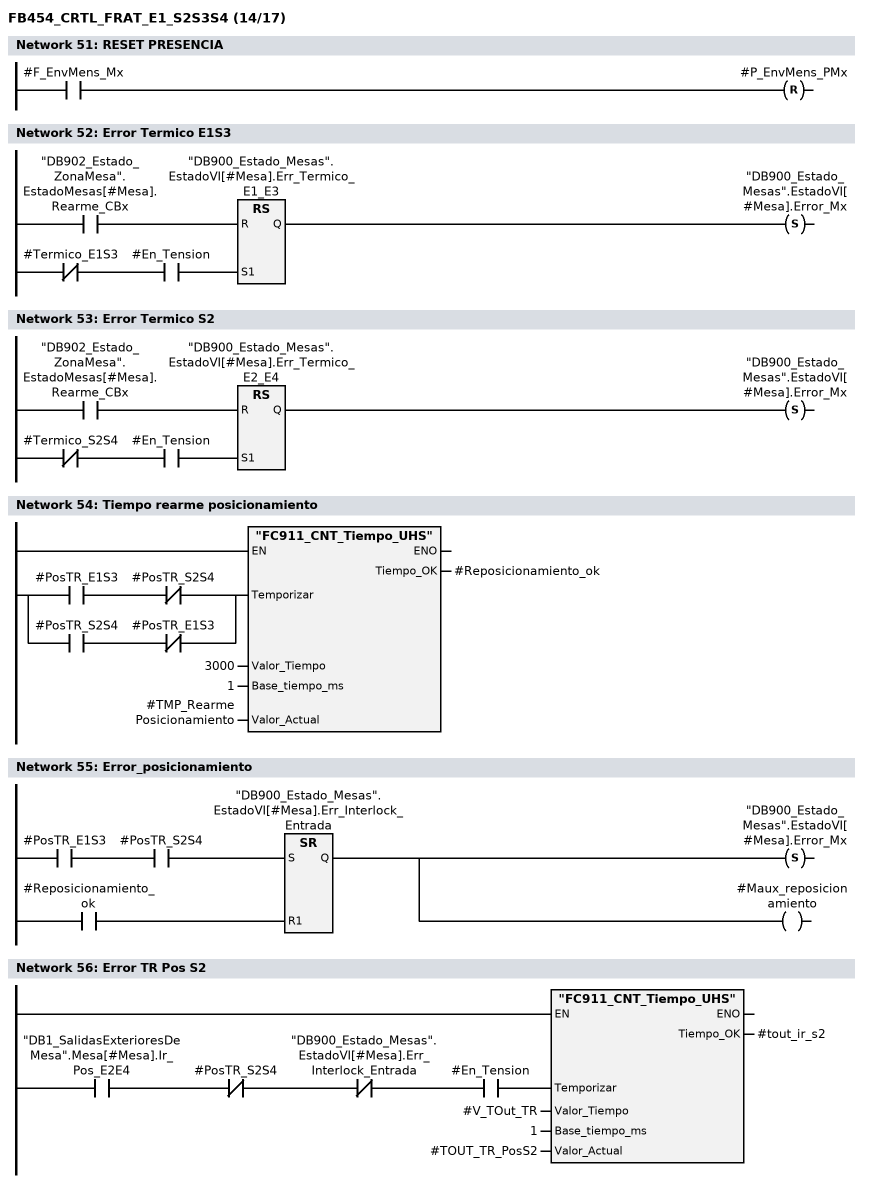
   RUNG wire#powerrail
      Contact( #F_EnvMens_Mx )
      R_Coil( #P_EnvMens_PMx )
   END_RUNG
   // the same network as SCL:
   IF #F_EnvMens_Mx THEN #P_EnvMens_PMx := FALSE; END_IF;
END_REGION

REGION Network 52: Error Termico E1S3
   RUNG wire#powerrail
      Contact( "DB902_Estado_ZonaMesa".EstadoMesas[#Mesa].Rearme_CBx )
      S_RS(operand := "DB900_Estado_Mesas".EstadoVI[#Mesa].Err_Termico_E1_E3, s1 := wire#w1)
      S_Coil( "DB900_Estado_Mesas".EstadoVI[#Mesa].Error_Mx )
   END_RUNG
   RUNG wire#powerrail
      I_Contact( #Termico_E1S3 )
      Contact( #En_Tension )
   END_RUNG wire#w1
   // the same network as SCL:
   IF "DB902_Estado_ZonaMesa".EstadoMesas[#Mesa].Rearme_CBx THEN
       "DB900_Estado_Mesas".EstadoVI[#Mesa].Err_Termico_E1_E3 := FALSE;   // RS flip-flop
   END_IF;
   IF NOT #Termico_E1S3 AND #En_Tension THEN
       "DB900_Estado_Mesas".EstadoVI[#Mesa].Err_Termico_E1_E3 := TRUE;
   END_IF;
   IF "DB900_Estado_Mesas".EstadoVI[#Mesa].Err_Termico_E1_E3 THEN
       "DB900_Estado_Mesas".EstadoVI[#Mesa].Error_Mx := TRUE;
   END_IF;
END_REGION

REGION Network 53: Error Termico S2
   RUNG wire#powerrail
      Contact( "DB902_Estado_ZonaMesa".EstadoMesas[#Mesa].Rearme_CBx )
      S_RS(operand := "DB900_Estado_Mesas".EstadoVI[#Mesa].Err_Termico_E2_E4, s1 := wire#w1)
      S_Coil( "DB900_Estado_Mesas".EstadoVI[#Mesa].Error_Mx )
   END_RUNG
   RUNG wire#powerrail
      I_Contact( #Termico_S2S4 )
      Contact( #En_Tension )
   END_RUNG wire#w1
   // the same network as SCL:
   IF "DB902_Estado_ZonaMesa".EstadoMesas[#Mesa].Rearme_CBx THEN
       "DB900_Estado_Mesas".EstadoVI[#Mesa].Err_Termico_E2_E4 := FALSE;   // RS flip-flop
   END_IF;
   IF NOT #Termico_S2S4 AND #En_Tension THEN
       "DB900_Estado_Mesas".EstadoVI[#Mesa].Err_Termico_E2_E4 := TRUE;
   END_IF;
   IF "DB900_Estado_Mesas".EstadoVI[#Mesa].Err_Termico_E2_E4 THEN
       "DB900_Estado_Mesas".EstadoVI[#Mesa].Error_Mx := TRUE;
   END_IF;
END_REGION

REGION Network 54: Tiempo rearme posicionamiento
   RUNG wire#powerrail
      "FC911_CNT_Tiempo_UHS"(Temporizar := wire#w1, Valor_Tiempo := 3000, Base_tiempo_ms := 1, Valor_Actual := #TMP_RearmePosicionamiento, Tiempo_OK => #Reposicionamiento_ok)
   END_RUNG
   RUNG wire#powerrail
      Contact( #PosTR_E1S3 )
      I_Contact( #PosTR_S2S4 )
   END_RUNG wire#w1
   RUNG wire#powerrail
      Contact( #PosTR_S2S4 )
      I_Contact( #PosTR_E1S3 )
   END_RUNG wire#w1
   // the same network as SCL:
   "FC911_CNT_Tiempo_UHS"(Temporizar := (#PosTR_E1S3 AND NOT #PosTR_S2S4) OR (#PosTR_S2S4 AND NOT #PosTR_E1S3),
                          Valor_Tiempo := 3000,
                          Base_tiempo_ms := 1,
                          Valor_Actual := #TMP_RearmePosicionamiento,
                          Tiempo_OK => #Reposicionamiento_ok);
END_REGION

REGION Network 55: Error_posicionamiento
   RUNG wire#powerrail
      Contact( #PosTR_E1S3 )
      Contact( #PosTR_S2S4 )
      S_SR(operand := "DB900_Estado_Mesas".EstadoVI[#Mesa].Err_Interlock_Entrada, r1 := wire#w1)
      wire#w2
      S_Coil( "DB900_Estado_Mesas".EstadoVI[#Mesa].Error_Mx )
   END_RUNG
   RUNG wire#powerrail
      Contact( #Reposicionamiento_ok )
   END_RUNG wire#w1
   RUNG wire#w2
      Coil( #Maux_reposicionamiento )
   END_RUNG
   // the same network as SCL:
   IF #PosTR_E1S3 AND #PosTR_S2S4 THEN
       "DB900_Estado_Mesas".EstadoVI[#Mesa].Err_Interlock_Entrada := TRUE;   // SR flip-flop
   END_IF;
   IF #Reposicionamiento_ok THEN "DB900_Estado_Mesas".EstadoVI[#Mesa].Err_Interlock_Entrada := FALSE; END_IF;
   #_w1 := "DB900_Estado_Mesas".EstadoVI[#Mesa].Err_Interlock_Entrada;
   IF #_w1 THEN "DB900_Estado_Mesas".EstadoVI[#Mesa].Error_Mx := TRUE; END_IF;
   #Maux_reposicionamiento := #_w1;
END_REGION

REGION Network 56: Error TR Pos S2
   RUNG wire#powerrail
      "FC911_CNT_Tiempo_UHS"(Temporizar := wire#w1, Valor_Tiempo := #V_TOut_TR, Base_tiempo_ms := 1, Valor_Actual := #TOUT_TR_PosS2, Tiempo_OK => #tout_ir_s2)
   END_RUNG
   RUNG wire#powerrail
      Contact( "DB1_SalidasExterioresDeMesa".Mesa[#Mesa].Ir_Pos_E2E4 )
      I_Contact( #PosTR_S2S4 )
      I_Contact( "DB900_Estado_Mesas".EstadoVI[#Mesa].Err_Interlock_Entrada )
      Contact( #En_Tension )
   END_RUNG wire#w1
   // the same network as SCL:
   "FC911_CNT_Tiempo_UHS"(Temporizar := "DB1_SalidasExterioresDeMesa".Mesa[#Mesa].Ir_Pos_E2E4 AND NOT #PosTR_S2S4 AND NOT "DB900_Estado_Mesas".EstadoVI[#Mesa].Err_Interlock_Entrada AND #En_Tension,
                          Valor_Tiempo := #V_TOut_TR,
                          Base_tiempo_ms := 1,
                          Valor_Actual := #TOUT_TR_PosS2,
                          Tiempo_OK => #tout_ir_s2);
END_REGION

REGION Network 57: ERROR TOUT SUBIDA TRANSFER
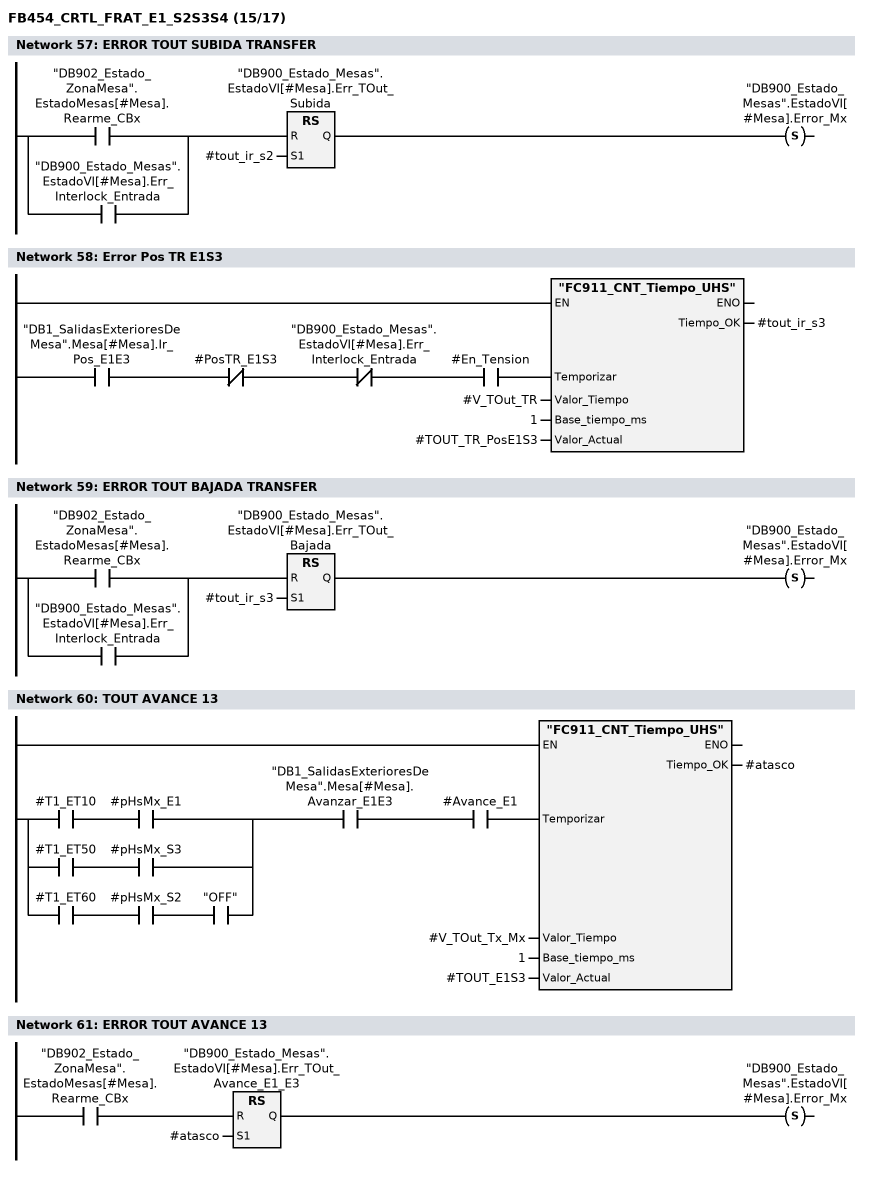
   RUNG wire#powerrail
      Contact( "DB902_Estado_ZonaMesa".EstadoMesas[#Mesa].Rearme_CBx )
      wire#w1
      S_RS(operand := "DB900_Estado_Mesas".EstadoVI[#Mesa].Err_TOut_Subida, s1 := #tout_ir_s2)
      S_Coil( "DB900_Estado_Mesas".EstadoVI[#Mesa].Error_Mx )
   END_RUNG
   RUNG wire#powerrail
      Contact( "DB900_Estado_Mesas".EstadoVI[#Mesa].Err_Interlock_Entrada )
   END_RUNG wire#w1
   // the same network as SCL:
   IF "DB902_Estado_ZonaMesa".EstadoMesas[#Mesa].Rearme_CBx OR "DB900_Estado_Mesas".EstadoVI[#Mesa].Err_Interlock_Entrada THEN
       "DB900_Estado_Mesas".EstadoVI[#Mesa].Err_TOut_Subida := FALSE;   // RS flip-flop
   END_IF;
   IF #tout_ir_s2 THEN "DB900_Estado_Mesas".EstadoVI[#Mesa].Err_TOut_Subida := TRUE; END_IF;
   IF "DB900_Estado_Mesas".EstadoVI[#Mesa].Err_TOut_Subida THEN
       "DB900_Estado_Mesas".EstadoVI[#Mesa].Error_Mx := TRUE;
   END_IF;
END_REGION

REGION Network 58: Error Pos TR E1S3
   RUNG wire#powerrail
      "FC911_CNT_Tiempo_UHS"(Temporizar := wire#w1, Valor_Tiempo := #V_TOut_TR, Base_tiempo_ms := 1, Valor_Actual := #TOUT_TR_PosE1S3, Tiempo_OK => #tout_ir_s3)
   END_RUNG
   RUNG wire#powerrail
      Contact( "DB1_SalidasExterioresDeMesa".Mesa[#Mesa].Ir_Pos_E1E3 )
      I_Contact( #PosTR_E1S3 )
      I_Contact( "DB900_Estado_Mesas".EstadoVI[#Mesa].Err_Interlock_Entrada )
      Contact( #En_Tension )
   END_RUNG wire#w1
   // the same network as SCL:
   "FC911_CNT_Tiempo_UHS"(Temporizar := "DB1_SalidasExterioresDeMesa".Mesa[#Mesa].Ir_Pos_E1E3 AND NOT #PosTR_E1S3 AND NOT "DB900_Estado_Mesas".EstadoVI[#Mesa].Err_Interlock_Entrada AND #En_Tension,
                          Valor_Tiempo := #V_TOut_TR,
                          Base_tiempo_ms := 1,
                          Valor_Actual := #TOUT_TR_PosE1S3,
                          Tiempo_OK => #tout_ir_s3);
END_REGION

REGION Network 59: ERROR TOUT BAJADA TRANSFER
   RUNG wire#powerrail
      Contact( "DB902_Estado_ZonaMesa".EstadoMesas[#Mesa].Rearme_CBx )
      wire#w1
      S_RS(operand := "DB900_Estado_Mesas".EstadoVI[#Mesa].Err_TOut_Bajada, s1 := #tout_ir_s3)
      S_Coil( "DB900_Estado_Mesas".EstadoVI[#Mesa].Error_Mx )
   END_RUNG
   RUNG wire#powerrail
      Contact( "DB900_Estado_Mesas".EstadoVI[#Mesa].Err_Interlock_Entrada )
   END_RUNG wire#w1
   // the same network as SCL:
   IF "DB902_Estado_ZonaMesa".EstadoMesas[#Mesa].Rearme_CBx OR "DB900_Estado_Mesas".EstadoVI[#Mesa].Err_Interlock_Entrada THEN
       "DB900_Estado_Mesas".EstadoVI[#Mesa].Err_TOut_Bajada := FALSE;   // RS flip-flop
   END_IF;
   IF #tout_ir_s3 THEN "DB900_Estado_Mesas".EstadoVI[#Mesa].Err_TOut_Bajada := TRUE; END_IF;
   IF "DB900_Estado_Mesas".EstadoVI[#Mesa].Err_TOut_Bajada THEN
       "DB900_Estado_Mesas".EstadoVI[#Mesa].Error_Mx := TRUE;
   END_IF;
END_REGION

REGION Network 60: TOUT AVANCE 13
   RUNG wire#powerrail
      "FC911_CNT_Tiempo_UHS"(Temporizar := wire#w2, Valor_Tiempo := #V_TOut_Tx_Mx, Base_tiempo_ms := 1, Valor_Actual := #TOUT_E1S3, Tiempo_OK => #atasco)
   END_RUNG
   RUNG wire#powerrail
      Contact( #T1_ET10 )
      Contact( #pHsMx_E1 )
      wire#w1
      Contact( "DB1_SalidasExterioresDeMesa".Mesa[#Mesa].Avanzar_E1E3 )
      Contact( #Avance_E1 )
   END_RUNG wire#w2
   RUNG wire#powerrail
      Contact( #T1_ET50 )
      Contact( #pHsMx_S3 )
   END_RUNG wire#w1
   RUNG wire#powerrail
      Contact( #T1_ET60 )
      Contact( #pHsMx_S2 )
      Contact( "OFF" )
   END_RUNG wire#w1
   // the same network as SCL:
   "FC911_CNT_Tiempo_UHS"(Temporizar := ((#T1_ET10 AND #pHsMx_E1) OR (#T1_ET50 AND #pHsMx_S3) OR (#T1_ET60 AND #pHsMx_S2 AND "OFF")) AND "DB1_SalidasExterioresDeMesa".Mesa[#Mesa].Avanzar_E1E3 AND #Avance_E1,
                          Valor_Tiempo := #V_TOut_Tx_Mx,
                          Base_tiempo_ms := 1,
                          Valor_Actual := #TOUT_E1S3,
                          Tiempo_OK => #atasco);
END_REGION

REGION Network 61: ERROR TOUT AVANCE 13
   RUNG wire#powerrail
      Contact( "DB902_Estado_ZonaMesa".EstadoMesas[#Mesa].Rearme_CBx )
      S_RS(operand := "DB900_Estado_Mesas".EstadoVI[#Mesa].Err_TOut_Avance_E1_E3, s1 := #atasco)
      S_Coil( "DB900_Estado_Mesas".EstadoVI[#Mesa].Error_Mx )
   END_RUNG
   // the same network as SCL:
   IF "DB902_Estado_ZonaMesa".EstadoMesas[#Mesa].Rearme_CBx THEN
       "DB900_Estado_Mesas".EstadoVI[#Mesa].Err_TOut_Avance_E1_E3 := FALSE;   // RS flip-flop
   END_IF;
   IF #atasco THEN "DB900_Estado_Mesas".EstadoVI[#Mesa].Err_TOut_Avance_E1_E3 := TRUE; END_IF;
   IF "DB900_Estado_Mesas".EstadoVI[#Mesa].Err_TOut_Avance_E1_E3 THEN
       "DB900_Estado_Mesas".EstadoVI[#Mesa].Error_Mx := TRUE;
   END_IF;
END_REGION

REGION Network 62: TOUT AVANCE S2
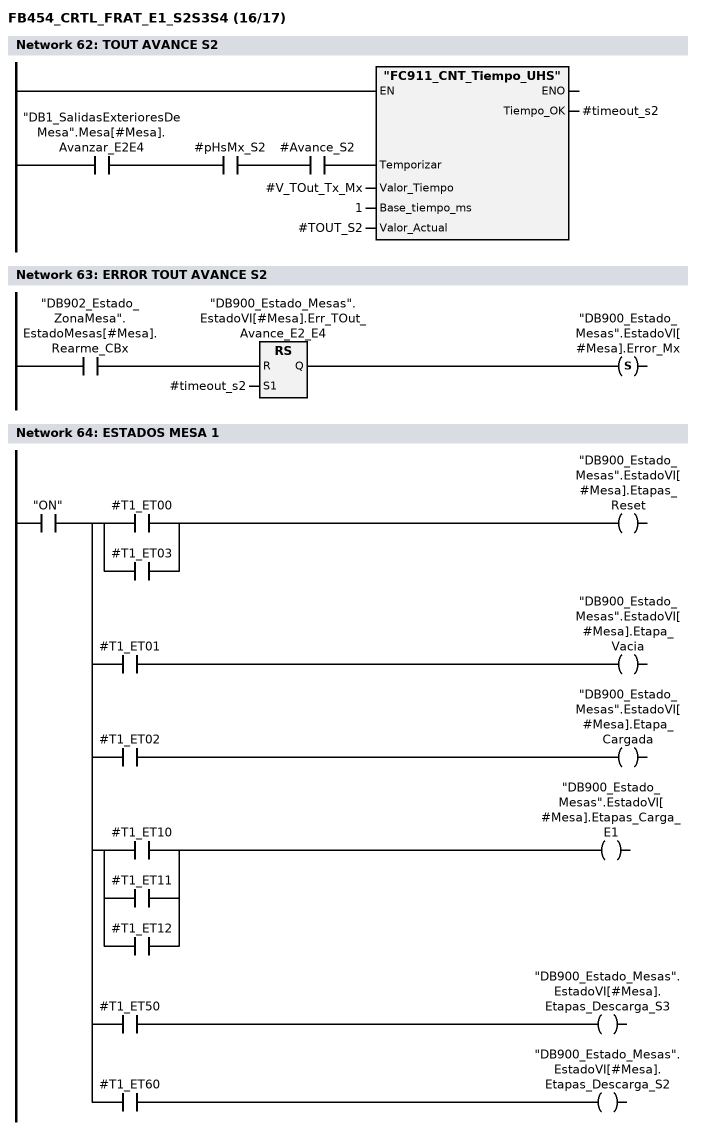
   RUNG wire#powerrail
      "FC911_CNT_Tiempo_UHS"(Temporizar := wire#w1, Valor_Tiempo := #V_TOut_Tx_Mx, Base_tiempo_ms := 1, Valor_Actual := #TOUT_S2, Tiempo_OK => #timeout_s2)
   END_RUNG
   RUNG wire#powerrail
      Contact( "DB1_SalidasExterioresDeMesa".Mesa[#Mesa].Avanzar_E2E4 )
      Contact( #pHsMx_S2 )
      Contact( #Avance_S2 )
   END_RUNG wire#w1
   // the same network as SCL:
   "FC911_CNT_Tiempo_UHS"(Temporizar := "DB1_SalidasExterioresDeMesa".Mesa[#Mesa].Avanzar_E2E4 AND #pHsMx_S2 AND #Avance_S2,
                          Valor_Tiempo := #V_TOut_Tx_Mx,
                          Base_tiempo_ms := 1,
                          Valor_Actual := #TOUT_S2,
                          Tiempo_OK => #timeout_s2);
END_REGION

REGION Network 63: ERROR TOUT AVANCE S2
   RUNG wire#powerrail
      Contact( "DB902_Estado_ZonaMesa".EstadoMesas[#Mesa].Rearme_CBx )
      S_RS(operand := "DB900_Estado_Mesas".EstadoVI[#Mesa].Err_TOut_Avance_E2_E4, s1 := #timeout_s2)
      S_Coil( "DB900_Estado_Mesas".EstadoVI[#Mesa].Error_Mx )
   END_RUNG
   // the same network as SCL:
   IF "DB902_Estado_ZonaMesa".EstadoMesas[#Mesa].Rearme_CBx THEN
       "DB900_Estado_Mesas".EstadoVI[#Mesa].Err_TOut_Avance_E2_E4 := FALSE;   // RS flip-flop
   END_IF;
   IF #timeout_s2 THEN "DB900_Estado_Mesas".EstadoVI[#Mesa].Err_TOut_Avance_E2_E4 := TRUE; END_IF;
   IF "DB900_Estado_Mesas".EstadoVI[#Mesa].Err_TOut_Avance_E2_E4 THEN
       "DB900_Estado_Mesas".EstadoVI[#Mesa].Error_Mx := TRUE;
   END_IF;
END_REGION

REGION Network 64: ESTADOS MESA 1
   RUNG wire#powerrail
      Contact( "ON" )
      wire#w1
      Contact( #T1_ET00 )
      wire#w2
      Coil( "DB900_Estado_Mesas".EstadoVI[#Mesa].Etapas_Reset )
   END_RUNG
   RUNG wire#w1
      Contact( #T1_ET03 )
   END_RUNG wire#w2
   RUNG wire#w1
      Contact( #T1_ET01 )
      Coil( "DB900_Estado_Mesas".EstadoVI[#Mesa].Etapa_Vacia )
   END_RUNG
   RUNG wire#w1
      Contact( #T1_ET02 )
      Coil( "DB900_Estado_Mesas".EstadoVI[#Mesa].Etapa_Cargada )
   END_RUNG
   RUNG wire#w1
      Contact( #T1_ET10 )
      wire#w3
      Coil( "DB900_Estado_Mesas".EstadoVI[#Mesa].Etapas_Carga_E1 )
   END_RUNG
   RUNG wire#w1
      Contact( #T1_ET11 )
   END_RUNG wire#w3
   RUNG wire#w1
      Contact( #T1_ET12 )
   END_RUNG wire#w3
   RUNG wire#w1
      Contact( #T1_ET50 )
      Coil( "DB900_Estado_Mesas".EstadoVI[#Mesa].Etapas_Descarga_S3 )
   END_RUNG
   RUNG wire#w1
      Contact( #T1_ET60 )
      Coil( "DB900_Estado_Mesas".EstadoVI[#Mesa].Etapas_Descarga_S2 )
   END_RUNG
   // the same network as SCL:
   "DB900_Estado_Mesas".EstadoVI[#Mesa].Etapas_Reset := "ON" AND (#T1_ET00 OR #T1_ET03);
   "DB900_Estado_Mesas".EstadoVI[#Mesa].Etapa_Vacia := "ON" AND #T1_ET01;
   "DB900_Estado_Mesas".EstadoVI[#Mesa].Etapa_Cargada := "ON" AND #T1_ET02;
   "DB900_Estado_Mesas".EstadoVI[#Mesa].Etapas_Carga_E1 := "ON" AND (#T1_ET10 OR #T1_ET11 OR #T1_ET12);
   "DB900_Estado_Mesas".EstadoVI[#Mesa].Etapas_Descarga_S3 := "ON" AND #T1_ET50;
   "DB900_Estado_Mesas".EstadoVI[#Mesa].Etapas_Descarga_S2 := "ON" AND #T1_ET60;
END_REGION

REGION Network 65: Entradas Mesas
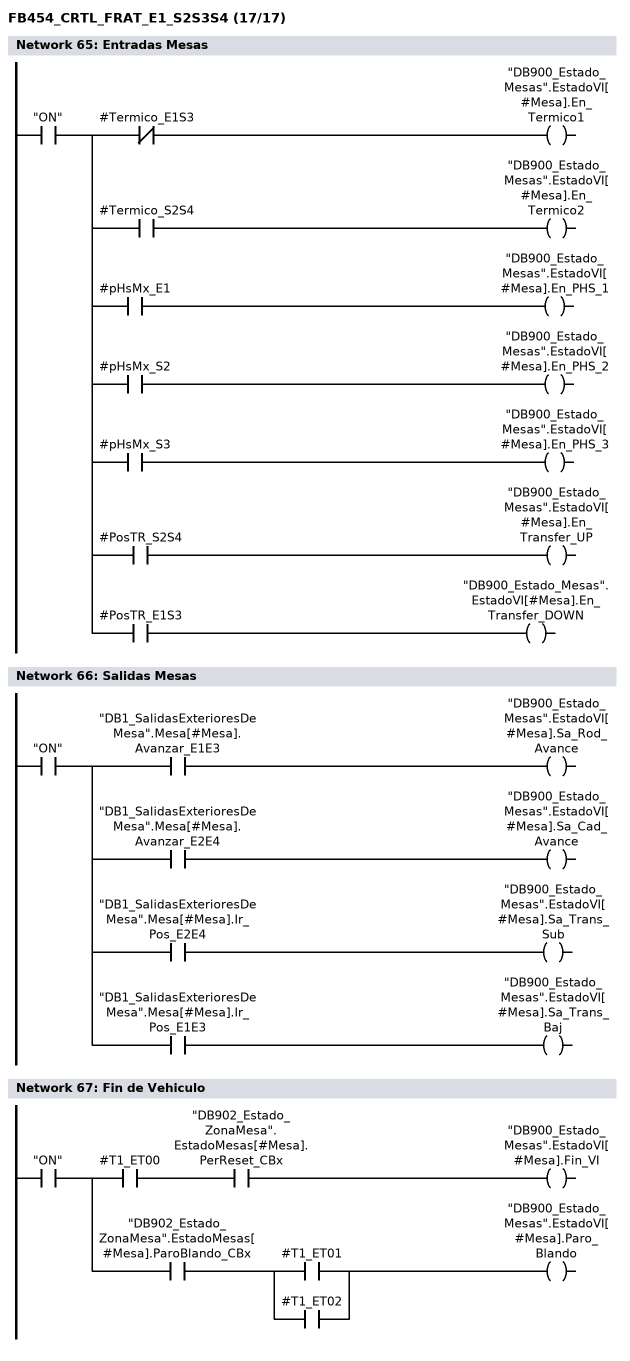
   RUNG wire#powerrail
      Contact( "ON" )
      wire#w1
      I_Contact( #Termico_E1S3 )
      Coil( "DB900_Estado_Mesas".EstadoVI[#Mesa].En_Termico1 )
   END_RUNG
   RUNG wire#w1
      Contact( #Termico_S2S4 )
      Coil( "DB900_Estado_Mesas".EstadoVI[#Mesa].En_Termico2 )
   END_RUNG
   RUNG wire#w1
      Contact( #pHsMx_E1 )
      Coil( "DB900_Estado_Mesas".EstadoVI[#Mesa].En_PHS_1 )
   END_RUNG
   RUNG wire#w1
      Contact( #pHsMx_S2 )
      Coil( "DB900_Estado_Mesas".EstadoVI[#Mesa].En_PHS_2 )
   END_RUNG
   RUNG wire#w1
      Contact( #pHsMx_S3 )
      Coil( "DB900_Estado_Mesas".EstadoVI[#Mesa].En_PHS_3 )
   END_RUNG
   RUNG wire#w1
      Contact( #PosTR_S2S4 )
      Coil( "DB900_Estado_Mesas".EstadoVI[#Mesa].En_Transfer_UP )
   END_RUNG
   RUNG wire#w1
      Contact( #PosTR_E1S3 )
      Coil( "DB900_Estado_Mesas".EstadoVI[#Mesa].En_Transfer_DOWN )
   END_RUNG
   // the same network as SCL:
   "DB900_Estado_Mesas".EstadoVI[#Mesa].En_Termico1 := "ON" AND NOT #Termico_E1S3;
   "DB900_Estado_Mesas".EstadoVI[#Mesa].En_Termico2 := "ON" AND #Termico_S2S4;
   "DB900_Estado_Mesas".EstadoVI[#Mesa].En_PHS_1 := "ON" AND #pHsMx_E1;
   "DB900_Estado_Mesas".EstadoVI[#Mesa].En_PHS_2 := "ON" AND #pHsMx_S2;
   "DB900_Estado_Mesas".EstadoVI[#Mesa].En_PHS_3 := "ON" AND #pHsMx_S3;
   "DB900_Estado_Mesas".EstadoVI[#Mesa].En_Transfer_UP := "ON" AND #PosTR_S2S4;
   "DB900_Estado_Mesas".EstadoVI[#Mesa].En_Transfer_DOWN := "ON" AND #PosTR_E1S3;
END_REGION

REGION Network 66: Salidas Mesas
   RUNG wire#powerrail
      Contact( "ON" )
      wire#w1
      Contact( "DB1_SalidasExterioresDeMesa".Mesa[#Mesa].Avanzar_E1E3 )
      Coil( "DB900_Estado_Mesas".EstadoVI[#Mesa].Sa_Rod_Avance )
   END_RUNG
   RUNG wire#w1
      Contact( "DB1_SalidasExterioresDeMesa".Mesa[#Mesa].Avanzar_E2E4 )
      Coil( "DB900_Estado_Mesas".EstadoVI[#Mesa].Sa_Cad_Avance )
   END_RUNG
   RUNG wire#w1
      Contact( "DB1_SalidasExterioresDeMesa".Mesa[#Mesa].Ir_Pos_E2E4 )
      Coil( "DB900_Estado_Mesas".EstadoVI[#Mesa].Sa_Trans_Sub )
   END_RUNG
   RUNG wire#w1
      Contact( "DB1_SalidasExterioresDeMesa".Mesa[#Mesa].Ir_Pos_E1E3 )
      Coil( "DB900_Estado_Mesas".EstadoVI[#Mesa].Sa_Trans_Baj )
   END_RUNG
   // the same network as SCL:
   "DB900_Estado_Mesas".EstadoVI[#Mesa].Sa_Rod_Avance := "ON" AND "DB1_SalidasExterioresDeMesa".Mesa[#Mesa].Avanzar_E1E3;
   "DB900_Estado_Mesas".EstadoVI[#Mesa].Sa_Cad_Avance := "ON" AND "DB1_SalidasExterioresDeMesa".Mesa[#Mesa].Avanzar_E2E4;
   "DB900_Estado_Mesas".EstadoVI[#Mesa].Sa_Trans_Sub := "ON" AND "DB1_SalidasExterioresDeMesa".Mesa[#Mesa].Ir_Pos_E2E4;
   "DB900_Estado_Mesas".EstadoVI[#Mesa].Sa_Trans_Baj := "ON" AND "DB1_SalidasExterioresDeMesa".Mesa[#Mesa].Ir_Pos_E1E3;
END_REGION

REGION Network 67: Fin de Vehiculo
   RUNG wire#powerrail
      Contact( "ON" )
      wire#w1
      Contact( #T1_ET00 )
      Contact( "DB902_Estado_ZonaMesa".EstadoMesas[#Mesa].PerReset_CBx )
      Coil( "DB900_Estado_Mesas".EstadoVI[#Mesa].Fin_VI )
   END_RUNG
   RUNG wire#w1
      Contact( "DB902_Estado_ZonaMesa".EstadoMesas[#Mesa].ParoBlando_CBx )
      wire#w2
      Contact( #T1_ET01 )
      wire#w3
      Coil( "DB900_Estado_Mesas".EstadoVI[#Mesa].Paro_Blando )
   END_RUNG
   RUNG wire#w2
      Contact( #T1_ET02 )
   END_RUNG wire#w3
   // the same network as SCL:
   "DB900_Estado_Mesas".EstadoVI[#Mesa].Fin_VI := "ON" AND #T1_ET00 AND "DB902_Estado_ZonaMesa".EstadoMesas[#Mesa].PerReset_CBx;
   "DB900_Estado_Mesas".EstadoVI[#Mesa].Paro_Blando := "ON" AND "DB902_Estado_ZonaMesa".EstadoMesas[#Mesa].ParoBlando_CBx AND (#T1_ET01 OR #T1_ET02);
END_REGION
END_FUNCTION_BLOCK
